(* CoDeSys 2.3 project: CX_KNX_TEST.pro *)
(* Title: BC and KL6301 *)
(* Version: 1.00 *)
(* Author: RV *)
(* Description: Demoproject for receive EIB Data
BC9000
KL6301
KL9010 *)
(* Libraries: TcpIp.lib 13.10.11 10:31:34, TcUtilities.lib 8.2.10 17:42:18, TcSocketHelper.lib 20.8.09 10:46:08, TcBase.lib 14.5.09 12:14:08, standard.lib 5.6.98 12:03:02, ClientStrSock.lib 19.10.12 18:01:27, TcSystem.lib 9.3.10 11:21:30, TcModbusSrv.lib 26.1.12 11:11:48, TcKL6301.lib 4.11.10 11:26:24 *)

(* Task configuration *)
TASK NeueTask (PRIORITY := 0, INTERVAL := T#10ms);
	MAIN();
END_TASK
TASK PowerCalc (PRIORITY := 2, INTERVAL := T#100ms);
	CalcPower();
END_TASK
TASK AdsSend (PRIORITY := 3, INTERVAL := T#1000ms);
	CheckLight();
END_TASK
TASK NewTask (PRIORITY := 1, INTERVAL := T#250ms);
	POWER_OFF_TEST();
	ReadADS();
END_TASK

(* Global variable list: Global_Variables_Power *)
VAR_GLOBAL

	KL3403_ctrl_1 AT%Q* : BYTE;

	KL3403_1_P1 AT%I* : INT;
	KL3403_1_P2 AT%I* : INT;
	KL3403_1_P3 AT%I* : INT;

	KL3403_1_P: REAL;
	KL3403_1_V: REAL;
	KL3403_1_I: REAL;

	KL3403_2_P1 AT%I* : INT;
	KL3403_2_P2 AT%I* : INT;
	KL3403_2_P3 AT%I* : INT;

	KL3403_2_P: REAL;
	KL3403_2_V: REAL;
	KL3403_2_I: REAL;

	KL3403_3_P1 AT%I* : INT;
	KL3403_3_P2 AT%I* : INT;
	KL3403_3_P3 AT%I* : INT;

	KL3403_3_P: REAL;
	KL3403_3_V: REAL;
	KL3403_3_I: REAL;

	KL3403_4_P1 AT%I* : INT;
	KL3403_4_P2 AT%I* : INT;
	KL3403_4_P3 AT%I* : INT;

	KL3403_4_P: REAL;
	KL3403_4_V: REAL;
	KL3403_4_I: REAL;

	KL3403_5_P1 AT%I* : INT;
	KL3403_5_P2 AT%I* : INT;
	KL3403_5_P3 AT%I* : INT;

	KL3403_5_P: REAL;
	KL3403_5_V: REAL;
	KL3403_5_I: REAL;

(*array of powers in VRU*)

(*
1 - schavp1		3
2 - schrd			11
3 - parouvl		2
4 - schnvd		5
5 - schrb			6
6 - schl			9
7 - schrov		1
8 - schss			10
9 - schuf			4
10 - schno		7
11 - hammam		8

7 - schrov		1
3 - parouvl		2
1 - schavp1		3
9 - schuf			4
4 - schnvd		5
5 - schrb			6
10 - schno		7
11 - hammam		8
6 - schl			9
8 - schss			10
2 - schrd			11

*)

	POWER_LIMIT: REAL;
	Current_switch_pos: INT;

	power_VRU_switch:  ARRAY[1..11] OF BOOL;
	(* priority*)
	power_VRU_address:  ARRAY[1..11] OF EIB_GROUP_ADDR;
	power_VRU_value: ARRAY[1..11] OF REAL;


	PowerSystemSwitcher: BOOL := TRUE;

END_VAR

(* Global variable list: Globale_Variablen *)
VAR_GLOBAL
    	bCloseAll 					: BOOL := TRUE;
   	bCreateSock					: BOOL := TRUE;

	ModByte			: BYTE;
	ModbusVentili	: BYTE;

	OutLightBytes		: BYTE;
	ControlLights		: BYTE;

	SCHAV			: ARRAY [1..4] OF INT;
	SCHNOG		: ARRAY [1..9] OF BOOL;

	schav_receive_stack AT %MB500 : ARRAY[1..7] OF INT;
	schav_force_stack AT %MB250 : ARRAY[1..7] OF INT;
	schnog_receive_stack AT %MB65 : ARRAY[1..19] OF BOOL;
	schnog_force_stack AT %MB265 : ARRAY[1..19] OF BOOL;
	schszp_receive_stack AT %MB100 : ARRAY[1..116] OF BOOL;
	schszp_force_stack AT %MB4500 : ARRAY[1..116] OF BOOL;
	(*tempMain_udp_packet AT %MB6000 : Udp_Packet;*)
	Main_udp_packet AT %MB2000 : Udp_Packet;
	Force_udp_packet AT %MB3000 : Udp_Packet;
	Temp_of_int AT %MB3006 : ARRAY[1..213] OF INT; (*область памяти совпадает с Force_udp_packet*)
	Confirmation_packet : Udp_Confirm;
	Received_packet AT %MB750 : Udp_Confirm;

	RESET_Edge : BOOL:=FALSE;
	TestWord : WORD;

	rByte : DINT;
	bSendConf : BOOL := FALSE;
	PacketSize: INT;
	Checksum_send : WORD;
	Checksum_incom : WORD;

	value3: INT;
	value2: INT;

	(*Считываем занчения вентиляторов*)
	CoolerByte		: BYTE;

	(* EIB terminal KL6301 process data 24 Byte input and 24 Byte output data K-Bus*)
	ShNOG_Garage_OG_22 AT %MB4 : BOOL:=FALSE;  (*Передаваемый параметр на другой контроллер. Свет в гараже - фуекция неисправного выхода модуля ABB KNX*)
	ShAV_Vent_V3 AT %MB5 : BOOL:=FALSE;  (*Передаваемый параметр на другой контроллер. Свет в туалете*)
	LightLandscape	: BOOL:=FALSE;  (*Передаваемый параметр на другой контроллер. Свет ландшафта*)
	LightNight AT %MB6 : BOOL := FALSE;  (*Передаваемый параметр на другой контроллер. "Ночь"*)
	KNXISDAY : BOOL := FALSE;
	KNXISTWILIGHT : BOOL := FALSE;
	LightNight_Clock AT %MB8 : BOOL := FALSE;

	SystemTime AT %MB4000 : TIMESTRUCT;
(*
	SS_H_AUT : WORD := 17; (*17*)
	SR_H_AUT : WORD := 6;
	SS_M_AUT : WORD := 19; (*19*)
	SR_M_AUT : WORD := 59;
	SS_H_WIN : WORD := 17; (*16*)
	SR_H_WIN : WORD := 8;
	SS_M_WIN : WORD := 19;
	SR_M_WIN : WORD := 29;
	SS_H_SPR : WORD := 19;
	SR_H_SPR : WORD := 5;
	SS_M_SPR : WORD := 19;
	SR_M_SPR : WORD := 29;
	SS_H_SUM : WORD := 21;
	SR_H_SUM : WORD := 4;
	SS_M_SUM : WORD := 01;
	SR_M_SUM : WORD := 01;
*)

	SS_H_JAN : WORD := 16;
	SR_H_JAN : WORD := 9;
	SS_M_JAN : WORD := 8;
	SR_M_JAN : WORD := 0;
	SS_H_FEB : WORD := 17;
	SR_H_FEB : WORD := 8;
	SS_M_FEB : WORD := 3;
	SR_M_FEB : WORD := 25;
	SS_H_MAR : WORD := 18;
	SR_H_MAR : WORD := 7;
	SS_M_MAR : WORD := 4;
	SR_M_MAR : WORD := 23;
	SS_H_APR : WORD := 19;
SR_H_APR : WORD := 6;
	SS_M_APR : WORD := 7;
SR_M_APR : WORD := 2;
	SS_H_MAY : WORD := 20;
SR_H_MAY : WORD := 4;
SS_M_MAY : WORD := 7;
SR_M_MAY : WORD := 48;
SS_H_JUN : WORD := 21;
SR_H_JUN : WORD := 3;
SS_M_JUN : WORD := 3;
SR_M_JUN : WORD := 55;
SS_H_JUL : WORD := 21;
SR_H_JUL : WORD := 3;
SS_M_JUL : WORD := 18;
SR_M_JUL : WORD := 51;
SS_H_AUG : WORD := 20;
SR_H_AUG : WORD := 4;
SS_M_AUG : WORD := 39;
SR_M_AUG : WORD := 35;
SS_H_SEP : WORD := 19;
SR_H_SEP : WORD := 5;
SS_M_SEP : WORD := 27;
SR_M_SEP : WORD := 35;
SS_H_OCT : WORD := 18;
SR_H_OCT : WORD := 6;
SS_M_OCT : WORD := 8;
SR_M_OCT : WORD := 33;
SS_H_NOV : WORD := 16;
SR_H_NOV : WORD := 7;
SS_M_NOV : WORD := 52;
SR_M_NOV : WORD := 36;
SS_H_DEC : WORD := 16;
SR_H_DEC : WORD := 8;
SS_M_DEC : WORD := 4;
SR_M_DEC : WORD := 36;

	JAN : WORD := 1;
	FEB : WORD := 2;
	MAR : WORD := 3;
	APR : WORD := 4;
	MAY : WORD := 5;
	JUN : WORD := 6;
	JUL : WORD := 7;
	AUG : WORD := 8;
	SEP : WORD := 9;
	OCT : WORD := 10;
	NOV : WORD := 11;
	DEC : WORD := 12;

	KNX_BRIGHTNESS_L : DINT;
	KNX_BRIGHTNESS_C : DINT;
	KNX_BRIGHTNESS_R : DINT;

	LightGarageSecurity : BOOL := FALSE;
	LightGatesLight AT %MB7 : BOOL:=FALSE;  (*Передаваемый параметр на другой контроллер. Выключатель света ворот в комнате охраны*)


	ADSSend: BOOL:=FALSE;

	KL6301_IN_0 AT %IB0: ARRAY[1..24] OF BYTE;
	KL6301_OUT_0 AT %QB0: ARRAY[1..24] OF BYTE;
	Taster0_LUX: BOOL;
	Taster1_LUX: BOOL;
	Taster2_LUX: BOOL;
	Taster3_LUX: BOOL;

	AllOff: BOOL;

	KoefV: BOOL:=FALSE;
	KoefI: BOOL:=FALSE;
	KoefP: BOOL:=TRUE;

	garage_OG_1: BOOL;
	garage_OG_2: BOOL;
	garage_OG_3: BOOL;
	garage_OG_4: BOOL;
	garage_OG_5: BOOL;
	garage_OG_6: BOOL;
	garage_OG_7: BOOL;
	garage_OG_8: BOOL;
	garage_OG_9: BOOL;
	garage_OG_10: BOOL;
	garage_OG_11: BOOL;
	garage_OG_12: BOOL;
	garage_OG_13: BOOL;
	garage_OG_14: BOOL;
	garage_OG_15: BOOL;
	garage_OG_16: BOOL;
	garage_OG_17: BOOL;
	garage_OG_18: BOOL;
	garage_OG_19: BOOL;
	garage_OG_20: BOOL;
	garage_OG_21: BOOL;
	garage_OG_22: BOOL;
	garage_OG_23: BOOL;
	garage_OG_24: BOOL;
	garage_OG_25: BOOL;
	garage_OG_26: BOOL;
	garage_OG_27: BOOL;
	garage_OG_28: BOOL;
	garage_OG_29: BOOL;

	SHUF_PRESSED: BOOL:= FALSE;

	DATA_SCALE_H									:INT :=255;
	DATA_SCALE_L									:INT :=0;
	DATA_SCALE_H_FAN								:INT :=32000;
	DATA_SCALE_L_FAN								:INT :=0;


END_VAR

VAR_GLOBAL CONSTANT
        TCPADS_MAXUDP_BUFFSIZE : UDINT :=32000;
END_VAR

(* Global variable list: Globale_Variablen_EIB *)
VAR_GLOBAL
	EIB_DATA_READ:  ARRAY[1..14] OF BYTE;
	Lux_REAL: REAL;	(* LUX *)
	Switch_0: BOOL;	(* Switch 1/2/1*)
	Switch_1: BOOL;	(* Switch 1/2/2*)
	Taster_0 AT %QX32.0: BOOL;
	Taster_1 AT %QX32.1: BOOL;
	Temp_0_KL3312 AT %IB26:INT;
	Temp_1_KL3312 AT %IB30:INT;
	IN_0_KL1012 AT %IX32.0:BOOL;
	IN_1_KL1012 AT %IX32.1:BOOL;
	str_Send: EIB_SEND;
	EIB_4FachT: BOOL;
	ToggleBit: BOOL;
	Soll_Lamp_Dimmer: INT;

	TurnAllTheLight: BOOL := FALSE;
END_VAR

(* Global variable list: TwinCAT_Configuration *)
(* Generated automatically by TwinCAT - (read only) *)
VAR_CONFIG
	.KL3403_ctrl_1 AT %QB36 : BYTE;	(*  ~ {LinkedWith:TIID^Device 3 (CX1100)^CX1100-KB^Term 2 (KL3403)^Channel 2^Ctrl;TIID^Device 3 (CX1100)^CX1100-KB^Term 2 (KL3403)^Channel 3^Ctrl;TIID^Device 3 (CX1100)^CX1100-KB^Term 3 (KL3403)^Channel 1^Ctrl;TIID^Device 3 (CX1100)^CX1100-KB^Term 3 (KL3403)^Channel 2^Ctrl;TIID^Device 3 (CX1100)^CX1100-KB^Term 3 (KL3403)^Channel 3^Ctrl;TIID^Device 3 (CX1100)^CX1100-KB^Term 4 (KL3403)^Channel 1^Ctrl;TIID^Device 3 (CX1100)^CX1100-KB^Term 4 (KL3403)^Channel 2^Ctrl;TIID^Device 3 (CX1100)^CX1100-KB^Term 4 (KL3403)^Channel 3^Ctrl;TIID^Device 3 (CX1100)^CX1100-KB^Term 5 (KL3403)^Channel 1^Ctrl;TIID^Device 3 (CX1100)^CX1100-KB^Term 5 (KL3403)^Channel 2^Ctrl;TIID^Device 3 (CX1100)^CX1100-KB^Term 5 (KL3403)^Channel 3^Ctrl;TIID^Device 3 (CX1100)^CX1100-KB^Term 6 (KL3403)^Channel 1^Ctrl;TIID^Device 3 (CX1100)^CX1100-KB^Term 6 (KL3403)^Channel 2^Ctrl;TIID^Device 3 (CX1100)^CX1100-KB^Term 6 (KL3403)^Channel 3^Ctrl;TIID^Device 3 (CX1100)^CX1100-KB^Term 2 (KL3403)^Channel 1^Ctrl} *)
	.KL3403_1_P1 AT %IB36 : INT;	(*  ~ {LinkedWith:TIID^Device 3 (CX1100)^CX1100-KB^Term 2 (KL3403)^Channel 1^Data In} *)
	.KL3403_1_P2 AT %IB38 : INT;	(*  ~ {LinkedWith:TIID^Device 3 (CX1100)^CX1100-KB^Term 2 (KL3403)^Channel 2^Data In} *)
	.KL3403_1_P3 AT %IB40 : INT;	(*  ~ {LinkedWith:TIID^Device 3 (CX1100)^CX1100-KB^Term 2 (KL3403)^Channel 3^Data In} *)
	.KL3403_2_P1 AT %IB42 : INT;	(*  ~ {LinkedWith:TIID^Device 3 (CX1100)^CX1100-KB^Term 3 (KL3403)^Channel 1^Data In} *)
	.KL3403_2_P2 AT %IB44 : INT;	(*  ~ {LinkedWith:TIID^Device 3 (CX1100)^CX1100-KB^Term 3 (KL3403)^Channel 2^Data In} *)
	.KL3403_2_P3 AT %IB46 : INT;	(*  ~ {LinkedWith:TIID^Device 3 (CX1100)^CX1100-KB^Term 3 (KL3403)^Channel 3^Data In} *)
	.KL3403_3_P1 AT %IB48 : INT;	(*  ~ {LinkedWith:TIID^Device 3 (CX1100)^CX1100-KB^Term 4 (KL3403)^Channel 1^Data In} *)
	.KL3403_3_P2 AT %IB50 : INT;	(*  ~ {LinkedWith:TIID^Device 3 (CX1100)^CX1100-KB^Term 4 (KL3403)^Channel 2^Data In} *)
	.KL3403_3_P3 AT %IB52 : INT;	(*  ~ {LinkedWith:TIID^Device 3 (CX1100)^CX1100-KB^Term 4 (KL3403)^Channel 3^Data In} *)
	.KL3403_4_P1 AT %IB54 : INT;	(*  ~ {LinkedWith:TIID^Device 3 (CX1100)^CX1100-KB^Term 5 (KL3403)^Channel 1^Data In} *)
	.KL3403_4_P2 AT %IB56 : INT;	(*  ~ {LinkedWith:TIID^Device 3 (CX1100)^CX1100-KB^Term 5 (KL3403)^Channel 2^Data In} *)
	.KL3403_4_P3 AT %IB58 : INT;	(*  ~ {LinkedWith:TIID^Device 3 (CX1100)^CX1100-KB^Term 5 (KL3403)^Channel 3^Data In} *)
	.KL3403_5_P1 AT %IB60 : INT;	(*  ~ {LinkedWith:TIID^Device 3 (CX1100)^CX1100-KB^Term 6 (KL3403)^Channel 1^Data In} *)
	.KL3403_5_P2 AT %IB62 : INT;	(*  ~ {LinkedWith:TIID^Device 3 (CX1100)^CX1100-KB^Term 6 (KL3403)^Channel 2^Data In} *)
	.KL3403_5_P3 AT %IB64 : INT;	(*  ~ {LinkedWith:TIID^Device 3 (CX1100)^CX1100-KB^Term 6 (KL3403)^Channel 3^Data In} *)
END_VAR

(* Data type *)
TYPE ST_FifoEntry :
STRUCT
	sRemoteHost		: STRING(15);		(* Remote address. String containing an (Ipv4) Internet Protocol dotted address. *)
	nRemotePort		: UDINT;			(* Remote Internet Protocol (IP) port. *)
	msg				: STRING;			(* Udp packet data *)
END_STRUCT
END_TYPE

(* Data type *)
TYPE Udp_Confirm :
STRUCT
	title_packet_num : INT;
	title_packet_code : INT;
	title_packet_crc : INT;
	data_pointer : INT;
	data_new_value : INT;
END_STRUCT
END_TYPE

(* Data type *)
TYPE Udp_Packet :
STRUCT
	title_packet_num : INT;
	title_packet_code : INT;
	title_packet_crc : INT;
	grsch_P : ARRAY[1..5] OF INT;
	grsch_V : ARRAY[1..5] OF INT;
	grsch_I : ARRAY[1..5] OF INT;
	grsch_garage_og : ARRAY[1..29] OF INT;
	grsch_power_VRU_value : ARRAY[1..11] OF INT;
	grsch_power_limit : INT;
	grsch_current_switch_pos : INT;
	grsch_power_VRU_switch : ARRAY[1..11] OF INT;
	grsch_SHUF_PRESSED : INT;
	grsch_power_system_switcher : INT;
	schav_stack : ARRAY[1..7] OF INT;
	schnog_stack : ARRAY[1..19] OF INT;
	schszp_stack  : ARRAY[1..116] OF INT;
END_STRUCT
END_TYPE

(* POU MAIN, ST *)
PROGRAM MAIN
VAR

	fbReadCoils : FB_MBReadCoils;
	bReadCoils : BOOL;
	nValue : BYTE;


	(* CX Controller *)
	(* KL6301 *)
	(* KL2xx2 *)
	(* KL9010 *)
	(* 1. EIB Device 2 Channel Switch Group Address 1/2/1 and 1 /2/2 *)
	(* 2. EIB Device Lux meter Group Address 1/1/5 *)
	fb_KL6301_0 : KL6301;	(* EIB functonblock *)
	i: INT := 0;				(* CASE *)
	EIB_DATA_SEND_0: EIB_SEND_DATA;
	fbTimer_0: TON;
	TimerOn: BOOL := FALSE;
	FLAG_01: BOOL := TRUE;
END_VAR
CASE i OF
0: 	fb_KL6301_0.bActivate :=FALSE; (*Start EIB Functionblock*)
	i := 1;

1:	fb_KL6301_0.EIB_PHYS_ADDR.Area:=2;		(* EIB Address 2.3.4 *)
	fb_KL6301_0.EIB_PHYS_ADDR.Line:=3;
	fb_KL6301_0.EIB_PHYS_ADDR.Device:=4;
	(* Filter 1 1/1/0 LEN 63*)
	fb_KL6301_0.EIB_GROUP_FILTER[1].GROUP_ADDR.MAIN:=1;
	fb_KL6301_0.EIB_GROUP_FILTER[1].GROUP_ADDR.SUB_MAIN:=1;
	fb_KL6301_0.EIB_GROUP_FILTER[1].GROUP_ADDR.NUMBER:=0;
	fb_KL6301_0.EIB_GROUP_FILTER[1].GROUP_LEN:=63;

	fb_KL6301_0.EIB_GROUP_FILTER[2].GROUP_ADDR.MAIN:=3;
	fb_KL6301_0.EIB_GROUP_FILTER[2].GROUP_ADDR.SUB_MAIN:=1;
	fb_KL6301_0.EIB_GROUP_FILTER[2].GROUP_ADDR.NUMBER:=0;
	fb_KL6301_0.EIB_GROUP_FILTER[2].GROUP_LEN:=63;

	fb_KL6301_0.EIB_GROUP_FILTER[3].GROUP_ADDR.MAIN:=5;
	fb_KL6301_0.EIB_GROUP_FILTER[3].GROUP_ADDR.SUB_MAIN:=1;
	fb_KL6301_0.EIB_GROUP_FILTER[3].GROUP_ADDR.NUMBER:=0;
	fb_KL6301_0.EIB_GROUP_FILTER[3].GROUP_LEN:=63;

	fb_KL6301_0.bActivate :=TRUE; (*Start EIB Functionblock*)

	IF fb_KL6301_0.bReady THEN
		IF NOT fb_KL6301_0.bError THEN
			i:=2;  (* EIB functionblock is now ready to send and receive *)
		ELSE
			i:=100; (* EIB ERROR*)
		END_IF
	END_IF
2:
(*Соберем всю инфу. По крайней мере, попробуем *)
KNX_Init;
(*POWER_OFF_TEST;*)

100:	;(*ERROR EIB*)
END_CASE

fb_KL6301_0(
	idx:=20,
	KL6301_IN:=KL6301_IN_0,				(* Terminal variable - address IN *)
	KL6301_OUT:=KL6301_OUT_0 );			(* Terminal variable - address OUT *)

Main_EIB_REC;

IF KoefV=TRUE THEN
	KL3403_ctrl_1:=1;
	KoefI:=FALSE;
	KoefV:=FALSE;
	KoefP:=FALSE;

END_IF

IF KoefI=TRUE THEN
	KL3403_ctrl_1:=0;
	KoefI:=FALSE;
	KoefV:=FALSE;
	KoefP:=FALSE;
END_IF

IF KoefP=TRUE THEN
	KL3403_ctrl_1:=2;
	KoefI:=FALSE;
	KoefV:=FALSE;
	KoefP:=FALSE;
END_IF

IF SHUF_PRESSED = TRUE THEN
	POWER_OFF_TEST;
	SHUF_PRESSED:= FALSE;
END_IF;

(* ZAPLATKA ZIMA VESNA LETO OSEN *)

IF (SystemTime.wMonth = JAN) AND SystemTime.wHour = SS_H_JAN AND SystemTime.wMinute = SS_M_JAN THEN
	LightNight_Clock := TRUE;						
END_IF;							
IF (SystemTime.wMonth = JAN) AND SystemTime.wHour = SR_H_JAN AND SystemTime.wMinute = SR_M_JAN THEN							
	LightNight_Clock := FALSE;						
END_IF;							
IF (SystemTime.wMonth = FEB) AND SystemTime.wHour = SS_H_FEB AND SystemTime.wMinute = SS_M_FEB THEN							
	LightNight_Clock := TRUE;						
END_IF;							
IF (SystemTime.wMonth = FEB) AND SystemTime.wHour = SR_H_FEB AND SystemTime.wMinute = SR_M_FEB THEN							
	LightNight_Clock := FALSE;						
END_IF;							
IF (SystemTime.wMonth = MAR) AND SystemTime.wHour = SS_H_MAR AND SystemTime.wMinute = SS_M_MAR THEN							
	LightNight_Clock := TRUE;						
END_IF;							
IF (SystemTime.wMonth = MAR) AND SystemTime.wHour = SR_H_MAR AND SystemTime.wMinute = SR_M_MAR THEN							
	LightNight_Clock := FALSE;						
END_IF;							
IF (SystemTime.wMonth = APR) AND SystemTime.wHour = SS_H_APR AND SystemTime.wMinute = SS_M_APR THEN							
	LightNight_Clock := TRUE;						
END_IF;							
IF (SystemTime.wMonth = APR) AND SystemTime.wHour = SR_H_APR AND SystemTime.wMinute = SR_M_APR THEN							
	LightNight_Clock := FALSE;						
END_IF;							
IF (SystemTime.wMonth = MAY) AND SystemTime.wHour = SS_H_MAY AND SystemTime.wMinute = SS_M_MAY THEN							
	LightNight_Clock := TRUE;						
END_IF;							
IF (SystemTime.wMonth = MAY) AND SystemTime.wHour = SR_H_MAY AND SystemTime.wMinute = SR_M_MAY THEN							
	LightNight_Clock := FALSE;						
END_IF;							
IF (SystemTime.wMonth = JUN) AND SystemTime.wHour = SS_H_JUN AND SystemTime.wMinute = SS_M_JUN THEN							
	LightNight_Clock := TRUE;						
END_IF;							
IF (SystemTime.wMonth = JUN) AND SystemTime.wHour = SR_H_JUN AND SystemTime.wMinute = SR_M_JUN THEN							
	LightNight_Clock := FALSE;						
END_IF;							
IF (SystemTime.wMonth = JUL) AND SystemTime.wHour = SS_H_JUL AND SystemTime.wMinute = SS_M_JUL THEN							
	LightNight_Clock := TRUE;						
END_IF;							
IF (SystemTime.wMonth = JUL) AND SystemTime.wHour = SR_H_JUL AND SystemTime.wMinute = SR_M_JUL THEN							
	LightNight_Clock := FALSE;						
END_IF;							
IF (SystemTime.wMonth = AUG) AND SystemTime.wHour = SS_H_AUG AND SystemTime.wMinute = SS_M_AUG THEN							
	LightNight_Clock := TRUE;						
END_IF;							
IF (SystemTime.wMonth = AUG) AND SystemTime.wHour = SR_H_AUG AND SystemTime.wMinute = SR_M_AUG THEN							
	LightNight_Clock := FALSE;						
END_IF;							
IF (SystemTime.wMonth = SEP) AND SystemTime.wHour = SS_H_SEP AND SystemTime.wMinute = SS_M_SEP THEN							
	LightNight_Clock := TRUE;						
END_IF;							
IF (SystemTime.wMonth = SEP) AND SystemTime.wHour = SR_H_SEP AND SystemTime.wMinute = SR_M_SEP THEN							
	LightNight_Clock := FALSE;						
END_IF;							
IF (SystemTime.wMonth = OCT) AND SystemTime.wHour = SS_H_OCT AND SystemTime.wMinute = SS_M_OCT THEN							
	LightNight_Clock := TRUE;						
END_IF;							
IF (SystemTime.wMonth = OCT) AND SystemTime.wHour = SR_H_OCT AND SystemTime.wMinute = SR_M_OCT THEN							
	LightNight_Clock := FALSE;						
END_IF;							
IF (SystemTime.wMonth = NOV) AND SystemTime.wHour = SS_H_NOV AND SystemTime.wMinute = SS_M_NOV THEN							
	LightNight_Clock := TRUE;						
END_IF;							
IF (SystemTime.wMonth = NOV) AND SystemTime.wHour = SR_H_NOV AND SystemTime.wMinute = SR_M_NOV THEN							
	LightNight_Clock := FALSE;						
END_IF;							
IF (SystemTime.wMonth = DEC) AND SystemTime.wHour = SS_H_DEC AND SystemTime.wMinute = SS_M_DEC THEN							
	LightNight_Clock := TRUE;						
END_IF;							
IF (SystemTime.wMonth = DEC) AND SystemTime.wHour = SR_H_DEC AND SystemTime.wMinute = SR_M_DEC THEN
	LightNight_Clock := FALSE;
END_IF;

(*
IF (SystemTime.wMonth = DEC OR SystemTime.wMonth = JAN OR SystemTime.wMonth = FEB) AND SystemTime.wHour = SS_H_WIN AND SystemTime.wMinute = SS_M_WIN THEN
	LightNight_Clock := TRUE;
END_IF;
IF (SystemTime.wMonth = DEC OR SystemTime.wMonth = JAN OR SystemTime.wMonth = FEB) AND SystemTime.wHour = SR_H_WIN AND SystemTime.wMinute = SR_M_WIN THEN
	LightNight_Clock := FALSE;
END_IF;

IF (SystemTime.wMonth = MAR OR SystemTime.wMonth = APR OR SystemTime.wMonth = MAY) AND SystemTime.wHour = SS_H_SPR AND SystemTime.wMinute = SS_M_SPR THEN
	LightNight_Clock := TRUE;
END_IF;
IF (SystemTime.wMonth = MAR OR SystemTime.wMonth = APR OR SystemTime.wMonth = MAY) AND SystemTime.wHour = SR_H_SPR AND SystemTime.wMinute = SR_M_SPR THEN
	LightNight_Clock := FALSE;
END_IF;

IF (SystemTime.wMonth = JUN OR SystemTime.wMonth = JUL OR SystemTime.wMonth = AUG) AND SystemTime.wHour = SS_H_SUM AND SystemTime.wMinute = SS_M_SUM THEN
	LightNight_Clock := TRUE;
END_IF;
IF (SystemTime.wMonth = JUN OR SystemTime.wMonth = JUL OR SystemTime.wMonth = AUG) AND SystemTime.wHour = SR_H_SUM AND SystemTime.wMinute = SR_M_SUM THEN
	LightNight_Clock := FALSE;
END_IF;

IF (SystemTime.wMonth = SEP OR SystemTime.wMonth = OCT OR SystemTime.wMonth = NOV) AND SystemTime.wHour = SS_H_AUT AND SystemTime.wMinute = SS_M_AUT THEN
	LightNight_Clock := TRUE;
END_IF;
IF (SystemTime.wMonth = SEP OR SystemTime.wMonth = OCT OR SystemTime.wMonth = NOV) AND SystemTime.wHour = SR_H_AUT AND SystemTime.wMinute = SR_M_AUT THEN
	LightNight_Clock := FALSE;
END_IF;

ZAPLATKA *)

IF KL6301_IN_0[10] = 16#0081 THEN
	LightGatesLight := TRUE;
ELSE
	LightGatesLight := FALSE;
END_IF;

Udp_send_packet_init;
PeerToPeer;
Udp_receive_packet_init;

IF (SystemTime.wDay = 15) AND SystemTime.wHour = 4 AND SystemTime.wMinute = 00 THEN
RESET_Edge:= TRUE;
AutoReset;
END_IF;
END_PROGRAM

(* POU KNX_Init, CFC *)
PROGRAM KNX_Init
VAR

(*свет*)
	Group_1_1_1: EIB_GROUP_ADDR := (MAIN:=1,SUB_MAIN:=1,NUMBER:=1);
	Group_1_1_2: EIB_GROUP_ADDR := (MAIN:=1,SUB_MAIN:=1,NUMBER:=2);
	Group_1_1_3: EIB_GROUP_ADDR := (MAIN:=1,SUB_MAIN:=1,NUMBER:=3);
	Group_1_1_4: EIB_GROUP_ADDR := (MAIN:=1,SUB_MAIN:=1,NUMBER:=4);
	Group_1_1_5: EIB_GROUP_ADDR := (MAIN:=1,SUB_MAIN:=1,NUMBER:=5);
	Group_1_1_6: EIB_GROUP_ADDR := (MAIN:=1,SUB_MAIN:=1,NUMBER:=6);
	Group_1_1_7: EIB_GROUP_ADDR := (MAIN:=1,SUB_MAIN:=1,NUMBER:=7);
	Group_1_1_8: EIB_GROUP_ADDR := (MAIN:=1,SUB_MAIN:=1,NUMBER:=8);
	Group_1_1_9: EIB_GROUP_ADDR := (MAIN:=1,SUB_MAIN:=1,NUMBER:=9);
	Group_1_1_10: EIB_GROUP_ADDR := (MAIN:=1,SUB_MAIN:=1,NUMBER:=10);
	Group_1_1_11: EIB_GROUP_ADDR := (MAIN:=1,SUB_MAIN:=1,NUMBER:=11);
	Group_1_1_12: EIB_GROUP_ADDR := (MAIN:=1,SUB_MAIN:=1,NUMBER:=12);
	Group_1_1_13: EIB_GROUP_ADDR := (MAIN:=1,SUB_MAIN:=1,NUMBER:=13);
	Group_1_1_14: EIB_GROUP_ADDR := (MAIN:=1,SUB_MAIN:=1,NUMBER:=14);
	Group_1_1_15: EIB_GROUP_ADDR := (MAIN:=1,SUB_MAIN:=1,NUMBER:=15);
	Group_1_1_16: EIB_GROUP_ADDR := (MAIN:=1,SUB_MAIN:=1,NUMBER:=16);
	Group_1_1_17: EIB_GROUP_ADDR := (MAIN:=1,SUB_MAIN:=1,NUMBER:=17);
	Group_1_1_18: EIB_GROUP_ADDR := (MAIN:=1,SUB_MAIN:=1,NUMBER:=18);
	Group_1_1_19: EIB_GROUP_ADDR := (MAIN:=1,SUB_MAIN:=1,NUMBER:=19);
	Group_1_1_20: EIB_GROUP_ADDR := (MAIN:=1,SUB_MAIN:=1,NUMBER:=20);
	Group_1_1_21: EIB_GROUP_ADDR := (MAIN:=1,SUB_MAIN:=1,NUMBER:=21);
	Group_1_1_22: EIB_GROUP_ADDR := (MAIN:=1,SUB_MAIN:=1,NUMBER:=22);
	Group_1_1_23: EIB_GROUP_ADDR := (MAIN:=1,SUB_MAIN:=1,NUMBER:=23);
	Group_1_1_24: EIB_GROUP_ADDR := (MAIN:=1,SUB_MAIN:=1,NUMBER:=24);
	Group_1_1_25: EIB_GROUP_ADDR := (MAIN:=1,SUB_MAIN:=1,NUMBER:=25);
	Group_1_1_26: EIB_GROUP_ADDR := (MAIN:=1,SUB_MAIN:=1,NUMBER:=26);
	Group_1_1_27: EIB_GROUP_ADDR := (MAIN:=1,SUB_MAIN:=1,NUMBER:=27);
	Group_1_1_28: EIB_GROUP_ADDR := (MAIN:=1,SUB_MAIN:=1,NUMBER:=28);
	Group_1_1_29: EIB_GROUP_ADDR := (MAIN:=1,SUB_MAIN:=1,NUMBER:=29);
	Group_1_1_30: EIB_GROUP_ADDR := (MAIN:=1,SUB_MAIN:=1,NUMBER:=30);
	Group_1_1_31: EIB_GROUP_ADDR := (MAIN:=1,SUB_MAIN:=1,NUMBER:=31);
	Group_1_1_32: EIB_GROUP_ADDR := (MAIN:=1,SUB_MAIN:=1,NUMBER:=32);
	Group_1_1_33: EIB_GROUP_ADDR := (MAIN:=1,SUB_MAIN:=1,NUMBER:=33);
	Group_1_1_34: EIB_GROUP_ADDR := (MAIN:=1,SUB_MAIN:=1,NUMBER:=34);
	Group_1_1_35: EIB_GROUP_ADDR := (MAIN:=1,SUB_MAIN:=1,NUMBER:=35);
	Group_1_1_36: EIB_GROUP_ADDR := (MAIN:=1,SUB_MAIN:=1,NUMBER:=36);
	Group_1_1_37: EIB_GROUP_ADDR := (MAIN:=1,SUB_MAIN:=1,NUMBER:=37);
	Group_1_1_38: EIB_GROUP_ADDR := (MAIN:=1,SUB_MAIN:=1,NUMBER:=38);
	KNXSYSTEM_WEATHERST_BRIGHTNES_L: EIB_GROUP_ADDR := (MAIN:=5,SUB_MAIN:=1,NUMBER:=2);
	KNXSYSTEM_WEATHERST_BRIGHTNES_C: EIB_GROUP_ADDR := (MAIN:=5,SUB_MAIN:=1,NUMBER:=3);
	KNXSYSTEM_WEATHERST_BRIGHTNES_R: EIB_GROUP_ADDR := (MAIN:=5,SUB_MAIN:=1,NUMBER:=4);
	KNXSYSTEM_WEATHERST_ISDAY: EIB_GROUP_ADDR := (MAIN:=5,SUB_MAIN:=1,NUMBER:=6);
	KNXSYSTEM_WEATHERST_ISTWILIGHT: EIB_GROUP_ADDR := (MAIN:=5,SUB_MAIN:=1,NUMBER:=40);

	init1: EIB_READ_SEND;
	init2: EIB_READ_SEND;
	init4: EIB_READ_SEND;
	init3: EIB_READ_SEND;
	init5: EIB_READ_SEND;
	init6: EIB_READ_SEND;
	init7: EIB_READ_SEND;
	init8: EIB_READ_SEND;
	init9: EIB_READ_SEND;
	init10: EIB_READ_SEND;
	init11: EIB_READ_SEND;
	init12: EIB_READ_SEND;
	init24: EIB_READ_SEND;
	init23: EIB_READ_SEND;
	init22: EIB_READ_SEND;
	init21: EIB_READ_SEND;
	init20: EIB_READ_SEND;
	init19: EIB_READ_SEND;
	init13: EIB_READ_SEND;
	init14: EIB_READ_SEND;
	init15: EIB_READ_SEND;
	init16: EIB_READ_SEND;
	init17: EIB_READ_SEND;
	init18: EIB_READ_SEND;
	init25: EIB_READ_SEND;
	init26: EIB_READ_SEND;
	init27: EIB_READ_SEND;
	init28: EIB_READ_SEND;
	init29: EIB_READ_SEND;
	init30: EIB_READ_SEND;
	init31: EIB_READ_SEND;
	init32: EIB_READ_SEND;
	init33: EIB_READ_SEND;
	init34: EIB_READ_SEND;
	init35: EIB_READ_SEND;
	init36: EIB_READ_SEND;
	init37: EIB_READ_SEND;
	init38: EIB_READ_SEND;
	init39: EIB_READ_SEND;
	init40: EIB_READ_SEND;
	init41: EIB_READ_SEND;
	init42: EIB_READ_SEND;
	init43: EIB_READ_SEND;
END_VAR
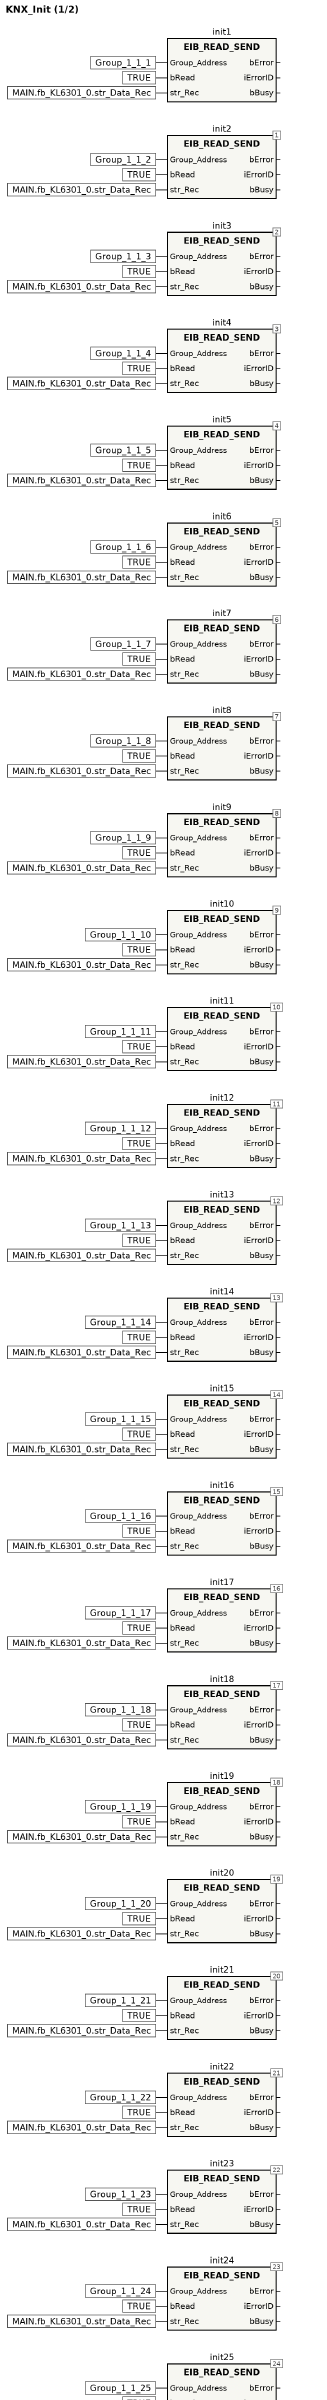
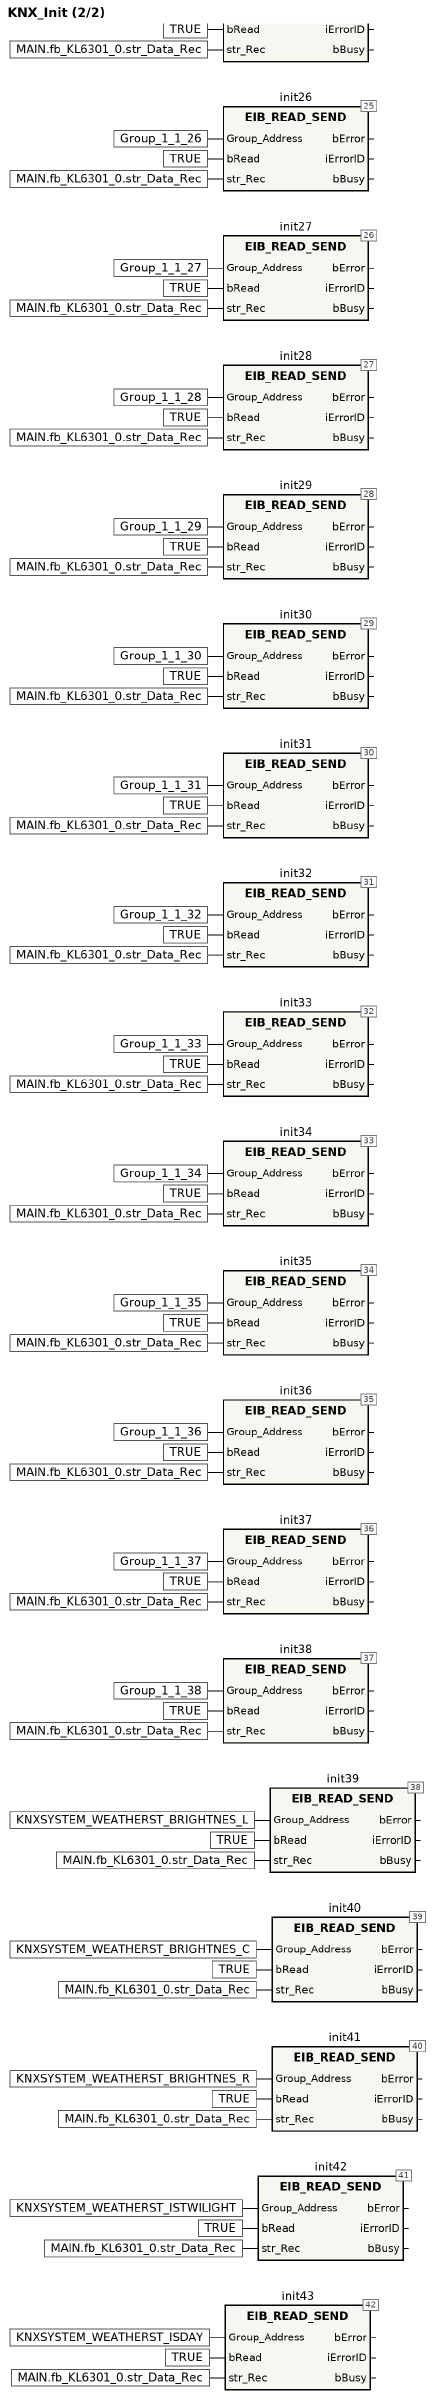
_CFC_ (* Continuous Function Chart, elements in execution order *)
#0 init1:EIB_READ_SEND(Group_Address: Group_1_1_1, bRead: TRUE, str_Rec: MAIN.fb_KL6301_0.str_Data_Rec)
#1 init2:EIB_READ_SEND(Group_Address: Group_1_1_2, bRead: TRUE, str_Rec: MAIN.fb_KL6301_0.str_Data_Rec)
#2 init3:EIB_READ_SEND(Group_Address: Group_1_1_3, bRead: TRUE, str_Rec: MAIN.fb_KL6301_0.str_Data_Rec)
#3 init4:EIB_READ_SEND(Group_Address: Group_1_1_4, bRead: TRUE, str_Rec: MAIN.fb_KL6301_0.str_Data_Rec)
#4 init5:EIB_READ_SEND(Group_Address: Group_1_1_5, bRead: TRUE, str_Rec: MAIN.fb_KL6301_0.str_Data_Rec)
#5 init6:EIB_READ_SEND(Group_Address: Group_1_1_6, bRead: TRUE, str_Rec: MAIN.fb_KL6301_0.str_Data_Rec)
#6 init7:EIB_READ_SEND(Group_Address: Group_1_1_7, bRead: TRUE, str_Rec: MAIN.fb_KL6301_0.str_Data_Rec)
#7 init8:EIB_READ_SEND(Group_Address: Group_1_1_8, bRead: TRUE, str_Rec: MAIN.fb_KL6301_0.str_Data_Rec)
#8 init9:EIB_READ_SEND(Group_Address: Group_1_1_9, bRead: TRUE, str_Rec: MAIN.fb_KL6301_0.str_Data_Rec)
#9 init10:EIB_READ_SEND(Group_Address: Group_1_1_10, bRead: TRUE, str_Rec: MAIN.fb_KL6301_0.str_Data_Rec)
#10 init11:EIB_READ_SEND(Group_Address: Group_1_1_11, bRead: TRUE, str_Rec: MAIN.fb_KL6301_0.str_Data_Rec)
#11 init12:EIB_READ_SEND(Group_Address: Group_1_1_12, bRead: TRUE, str_Rec: MAIN.fb_KL6301_0.str_Data_Rec)
#12 init13:EIB_READ_SEND(Group_Address: Group_1_1_13, bRead: TRUE, str_Rec: MAIN.fb_KL6301_0.str_Data_Rec)
#13 init14:EIB_READ_SEND(Group_Address: Group_1_1_14, bRead: TRUE, str_Rec: MAIN.fb_KL6301_0.str_Data_Rec)
#14 init15:EIB_READ_SEND(Group_Address: Group_1_1_15, bRead: TRUE, str_Rec: MAIN.fb_KL6301_0.str_Data_Rec)
#15 init16:EIB_READ_SEND(Group_Address: Group_1_1_16, bRead: TRUE, str_Rec: MAIN.fb_KL6301_0.str_Data_Rec)
#16 init17:EIB_READ_SEND(Group_Address: Group_1_1_17, bRead: TRUE, str_Rec: MAIN.fb_KL6301_0.str_Data_Rec)
#17 init18:EIB_READ_SEND(Group_Address: Group_1_1_18, bRead: TRUE, str_Rec: MAIN.fb_KL6301_0.str_Data_Rec)
#18 init19:EIB_READ_SEND(Group_Address: Group_1_1_19, bRead: TRUE, str_Rec: MAIN.fb_KL6301_0.str_Data_Rec)
#19 init20:EIB_READ_SEND(Group_Address: Group_1_1_20, bRead: TRUE, str_Rec: MAIN.fb_KL6301_0.str_Data_Rec)
#20 init21:EIB_READ_SEND(Group_Address: Group_1_1_21, bRead: TRUE, str_Rec: MAIN.fb_KL6301_0.str_Data_Rec)
#21 init22:EIB_READ_SEND(Group_Address: Group_1_1_22, bRead: TRUE, str_Rec: MAIN.fb_KL6301_0.str_Data_Rec)
#22 init23:EIB_READ_SEND(Group_Address: Group_1_1_23, bRead: TRUE, str_Rec: MAIN.fb_KL6301_0.str_Data_Rec)
#23 init24:EIB_READ_SEND(Group_Address: Group_1_1_24, bRead: TRUE, str_Rec: MAIN.fb_KL6301_0.str_Data_Rec)
#24 init25:EIB_READ_SEND(Group_Address: Group_1_1_25, bRead: TRUE, str_Rec: MAIN.fb_KL6301_0.str_Data_Rec)
#25 init26:EIB_READ_SEND(Group_Address: Group_1_1_26, bRead: TRUE, str_Rec: MAIN.fb_KL6301_0.str_Data_Rec)
#26 init27:EIB_READ_SEND(Group_Address: Group_1_1_27, bRead: TRUE, str_Rec: MAIN.fb_KL6301_0.str_Data_Rec)
#27 init28:EIB_READ_SEND(Group_Address: Group_1_1_28, bRead: TRUE, str_Rec: MAIN.fb_KL6301_0.str_Data_Rec)
#28 init29:EIB_READ_SEND(Group_Address: Group_1_1_29, bRead: TRUE, str_Rec: MAIN.fb_KL6301_0.str_Data_Rec)
#29 init30:EIB_READ_SEND(Group_Address: Group_1_1_30, bRead: TRUE, str_Rec: MAIN.fb_KL6301_0.str_Data_Rec)
#30 init31:EIB_READ_SEND(Group_Address: Group_1_1_31, bRead: TRUE, str_Rec: MAIN.fb_KL6301_0.str_Data_Rec)
#31 init32:EIB_READ_SEND(Group_Address: Group_1_1_32, bRead: TRUE, str_Rec: MAIN.fb_KL6301_0.str_Data_Rec)
#32 init33:EIB_READ_SEND(Group_Address: Group_1_1_33, bRead: TRUE, str_Rec: MAIN.fb_KL6301_0.str_Data_Rec)
#33 init34:EIB_READ_SEND(Group_Address: Group_1_1_34, bRead: TRUE, str_Rec: MAIN.fb_KL6301_0.str_Data_Rec)
#34 init35:EIB_READ_SEND(Group_Address: Group_1_1_35, bRead: TRUE, str_Rec: MAIN.fb_KL6301_0.str_Data_Rec)
#35 init36:EIB_READ_SEND(Group_Address: Group_1_1_36, bRead: TRUE, str_Rec: MAIN.fb_KL6301_0.str_Data_Rec)
#36 init37:EIB_READ_SEND(Group_Address: Group_1_1_37, bRead: TRUE, str_Rec: MAIN.fb_KL6301_0.str_Data_Rec)
#37 init38:EIB_READ_SEND(Group_Address: Group_1_1_38, bRead: TRUE, str_Rec: MAIN.fb_KL6301_0.str_Data_Rec)
#38 init39:EIB_READ_SEND(Group_Address: KNXSYSTEM_WEATHERST_BRIGHTNES_L, bRead: TRUE, str_Rec: MAIN.fb_KL6301_0.str_Data_Rec)
#39 init40:EIB_READ_SEND(Group_Address: KNXSYSTEM_WEATHERST_BRIGHTNES_C, bRead: TRUE, str_Rec: MAIN.fb_KL6301_0.str_Data_Rec)
#40 init41:EIB_READ_SEND(Group_Address: KNXSYSTEM_WEATHERST_BRIGHTNES_R, bRead: TRUE, str_Rec: MAIN.fb_KL6301_0.str_Data_Rec)
#41 init42:EIB_READ_SEND(Group_Address: KNXSYSTEM_WEATHERST_ISTWILIGHT, bRead: TRUE, str_Rec: MAIN.fb_KL6301_0.str_Data_Rec)
#42 init43:EIB_READ_SEND(Group_Address: KNXSYSTEM_WEATHERST_ISDAY, bRead: TRUE, str_Rec: MAIN.fb_KL6301_0.str_Data_Rec)
_END_CFC_
END_PROGRAM

(* POU Main_EIB_REC, CFC *)
PROGRAM Main_EIB_REC
VAR
	EIB_BIT_REC_0: EIB_BIT_REC;

(*	EIB_BIT_REC_1: EIB_BIT_REC;
	EIB_REAL_REC_0:EIB_2OCTET_FLOAT_REC;
	EIB_REAL_REC_Temp:EIB_2OCTET_FLOAT_REC;
	EIB_8Bit:EIB_8BIT_SIGN_REC;
	EIB_3Bit:EIB_3BIT_CONTROL_REC;
	EIB_3Bit_1:EIB_3BIT_CONTROL_REC;
	EIB_2BYTE_UINT:EIB_2OCTET_UNSIGN_REC;
	EIB_4UDINT:EIB_4OCTET_SIGN_REC;
	EIB_4Float:EIB_4OCTET_FLOAT_REC;  *)

	Group_1_1_1: EIB_GROUP_ADDR := (MAIN:=1,SUB_MAIN:=1,NUMBER:=1);
	Group_1_1_2: EIB_GROUP_ADDR := (MAIN:=1,SUB_MAIN:=1,NUMBER:=2);
	Group_1_1_3: EIB_GROUP_ADDR := (MAIN:=1,SUB_MAIN:=1,NUMBER:=3);
	Group_1_1_4: EIB_GROUP_ADDR := (MAIN:=1,SUB_MAIN:=1,NUMBER:=4);
	Group_1_1_5: EIB_GROUP_ADDR := (MAIN:=1,SUB_MAIN:=1,NUMBER:=5);
	Group_1_1_6: EIB_GROUP_ADDR := (MAIN:=1,SUB_MAIN:=1,NUMBER:=6);
	Group_1_1_7: EIB_GROUP_ADDR := (MAIN:=1,SUB_MAIN:=1,NUMBER:=7);
	Group_1_1_8: EIB_GROUP_ADDR := (MAIN:=1,SUB_MAIN:=1,NUMBER:=8);
	Group_1_1_9: EIB_GROUP_ADDR := (MAIN:=1,SUB_MAIN:=1,NUMBER:=9);
	Group_1_1_10: EIB_GROUP_ADDR := (MAIN:=1,SUB_MAIN:=1,NUMBER:=10);
	Group_1_1_11: EIB_GROUP_ADDR := (MAIN:=1,SUB_MAIN:=1,NUMBER:=11);
	Group_1_1_12: EIB_GROUP_ADDR := (MAIN:=1,SUB_MAIN:=1,NUMBER:=12);
	Group_1_1_13: EIB_GROUP_ADDR := (MAIN:=1,SUB_MAIN:=1,NUMBER:=13);
	Group_1_1_14: EIB_GROUP_ADDR := (MAIN:=1,SUB_MAIN:=1,NUMBER:=14);
	Group_1_1_15: EIB_GROUP_ADDR := (MAIN:=1,SUB_MAIN:=1,NUMBER:=15);
	Group_1_1_16: EIB_GROUP_ADDR := (MAIN:=1,SUB_MAIN:=1,NUMBER:=16);
	Group_1_1_17: EIB_GROUP_ADDR := (MAIN:=1,SUB_MAIN:=1,NUMBER:=17);
	Group_1_1_18: EIB_GROUP_ADDR := (MAIN:=1,SUB_MAIN:=1,NUMBER:=18);
	Group_1_1_19: EIB_GROUP_ADDR := (MAIN:=1,SUB_MAIN:=1,NUMBER:=19);
	Group_1_1_20: EIB_GROUP_ADDR := (MAIN:=1,SUB_MAIN:=1,NUMBER:=20);
	Group_1_1_21: EIB_GROUP_ADDR := (MAIN:=1,SUB_MAIN:=1,NUMBER:=21);
	Group_1_1_22: EIB_GROUP_ADDR := (MAIN:=1,SUB_MAIN:=1,NUMBER:=22);
	Group_1_1_23: EIB_GROUP_ADDR := (MAIN:=1,SUB_MAIN:=1,NUMBER:=23);
	Group_1_1_24: EIB_GROUP_ADDR := (MAIN:=1,SUB_MAIN:=1,NUMBER:=24);
	Group_1_1_25: EIB_GROUP_ADDR := (MAIN:=1,SUB_MAIN:=1,NUMBER:=25);
	Group_1_1_26: EIB_GROUP_ADDR := (MAIN:=1,SUB_MAIN:=1,NUMBER:=26);
	Group_1_1_27: EIB_GROUP_ADDR := (MAIN:=1,SUB_MAIN:=1,NUMBER:=27);
	Group_1_1_28: EIB_GROUP_ADDR := (MAIN:=1,SUB_MAIN:=1,NUMBER:=28);
	Group_1_1_29: EIB_GROUP_ADDR := (MAIN:=1,SUB_MAIN:=1,NUMBER:=29);  (*zdes bilo MAIN:=5,SUB_MAIN:=1,NUMBER:=6. Sozdal otdelnuyu peremennuyu s etim adresom nizhe*)
	Group_1_1_30: EIB_GROUP_ADDR := (MAIN:=1,SUB_MAIN:=1,NUMBER:=30);

	Group_1_1_31: EIB_GROUP_ADDR := (MAIN:=1,SUB_MAIN:=1,NUMBER:=31);
	Group_1_1_32: EIB_GROUP_ADDR := (MAIN:=1,SUB_MAIN:=1,NUMBER:=32);
	Group_1_1_33: EIB_GROUP_ADDR := (MAIN:=1,SUB_MAIN:=1,NUMBER:=33);
	Group_1_1_34: EIB_GROUP_ADDR := (MAIN:=1,SUB_MAIN:=1,NUMBER:=34);
	Group_1_1_35: EIB_GROUP_ADDR := (MAIN:=1,SUB_MAIN:=1,NUMBER:=35);
	Group_1_1_36: EIB_GROUP_ADDR := (MAIN:=1,SUB_MAIN:=1,NUMBER:=36);
	Group_1_1_37: EIB_GROUP_ADDR := (MAIN:=1,SUB_MAIN:=1,NUMBER:=37);
	Group_1_1_38: EIB_GROUP_ADDR := (MAIN:=1,SUB_MAIN:=1,NUMBER:=38);

	KNXSYSTEM_WEATHERST_BRIGHTNES_L: EIB_GROUP_ADDR := (MAIN:=5,SUB_MAIN:=1,NUMBER:=2);
	KNXSYSTEM_WEATHERST_BRIGHTNES_C: EIB_GROUP_ADDR := (MAIN:=5,SUB_MAIN:=1,NUMBER:=3);
	KNXSYSTEM_WEATHERST_BRIGHTNES_R: EIB_GROUP_ADDR := (MAIN:=5,SUB_MAIN:=1,NUMBER:=4);
	KNXSYSTEM_WEATHERST_ISTWILIGHT: EIB_GROUP_ADDR := (MAIN:=5,SUB_MAIN:=1,NUMBER:=40);
	KNXSYSTEM_WEATHERST_ISDAY: EIB_GROUP_ADDR := (MAIN:=5,SUB_MAIN:=1,NUMBER:=6);

	EIB_BIT_REC_1: EIB_BIT_REC;
	EIB_BIT_REC_2: EIB_BIT_REC;
	EIB_BIT_REC_3: EIB_BIT_REC;
	EIB_BIT_REC_4: EIB_BIT_REC;
	EIB_BIT_REC_5: EIB_BIT_REC;
	EIB_BIT_REC_6: EIB_BIT_REC;
	EIB_BIT_REC_7: EIB_BIT_REC;
	EIB_BIT_REC_8: EIB_BIT_REC;
	EIB_BIT_REC_9: EIB_BIT_REC;
	EIB_BIT_REC_10: EIB_BIT_REC;
	EIB_BIT_REC_11: EIB_BIT_REC;
	EIB_BIT_REC_12: EIB_BIT_REC;
	EIB_BIT_REC_13: EIB_BIT_REC;
	EIB_BIT_REC_14: EIB_BIT_REC;
	EIB_BIT_REC_15: EIB_BIT_REC;
	EIB_BIT_REC_16: EIB_BIT_REC;
	EIB_BIT_REC_17: EIB_BIT_REC;
	EIB_BIT_REC_18: EIB_BIT_REC;
	EIB_BIT_REC_19: EIB_BIT_REC;
	EIB_BIT_REC_20: EIB_BIT_REC;
	EIB_BIT_REC_21: EIB_BIT_REC;
	EIB_BIT_REC_22: EIB_BIT_REC;
	EIB_BIT_REC_23: EIB_BIT_REC;
	EIB_BIT_REC_24: EIB_BIT_REC;
	EIB_BIT_REC_25: EIB_BIT_REC;
	EIB_BIT_REC_26: EIB_BIT_REC;
	EIB_BIT_REC_27: EIB_BIT_REC;
	EIB_BIT_REC_28: EIB_BIT_REC;
	EIB_BIT_REC_29: EIB_BIT_REC;
	EIB_BIT_REC_30: EIB_BIT_REC;
	EIB_BIT_REC_31: EIB_BIT_REC;
	EIB_BIT_REC_32: EIB_BIT_REC;
	EIB_BIT_REC_33: EIB_BIT_REC;
	EIB_BIT_REC_34: EIB_BIT_REC;
	EIB_BIT_REC_35: EIB_BIT_REC;
	EIB_BIT_REC_36: EIB_BIT_REC;
	EIB_BIT_REC_37: EIB_BIT_REC;
	EIB_BIT_REC_38: EIB_BIT_REC;
	EIB_BIT_REC_39: EIB_BIT_REC;
	EIB_BIT_REC_40: EIB_BIT_REC;
	EIB_BIT_REC_41: EIB_BIT_REC;
	EIB_ALL_DATA_TYPES_REC_40: EIB_4OCTET_SIGN_REC;
	EIB_ALL_DATA_TYPES_REC_41: EIB_4OCTET_SIGN_REC;
	EIB_ALL_DATA_TYPES_REC_42: EIB_4OCTET_SIGN_REC;
	fb_GetTi: NT_GetTime;
	Timer1: TON;
END_VAR
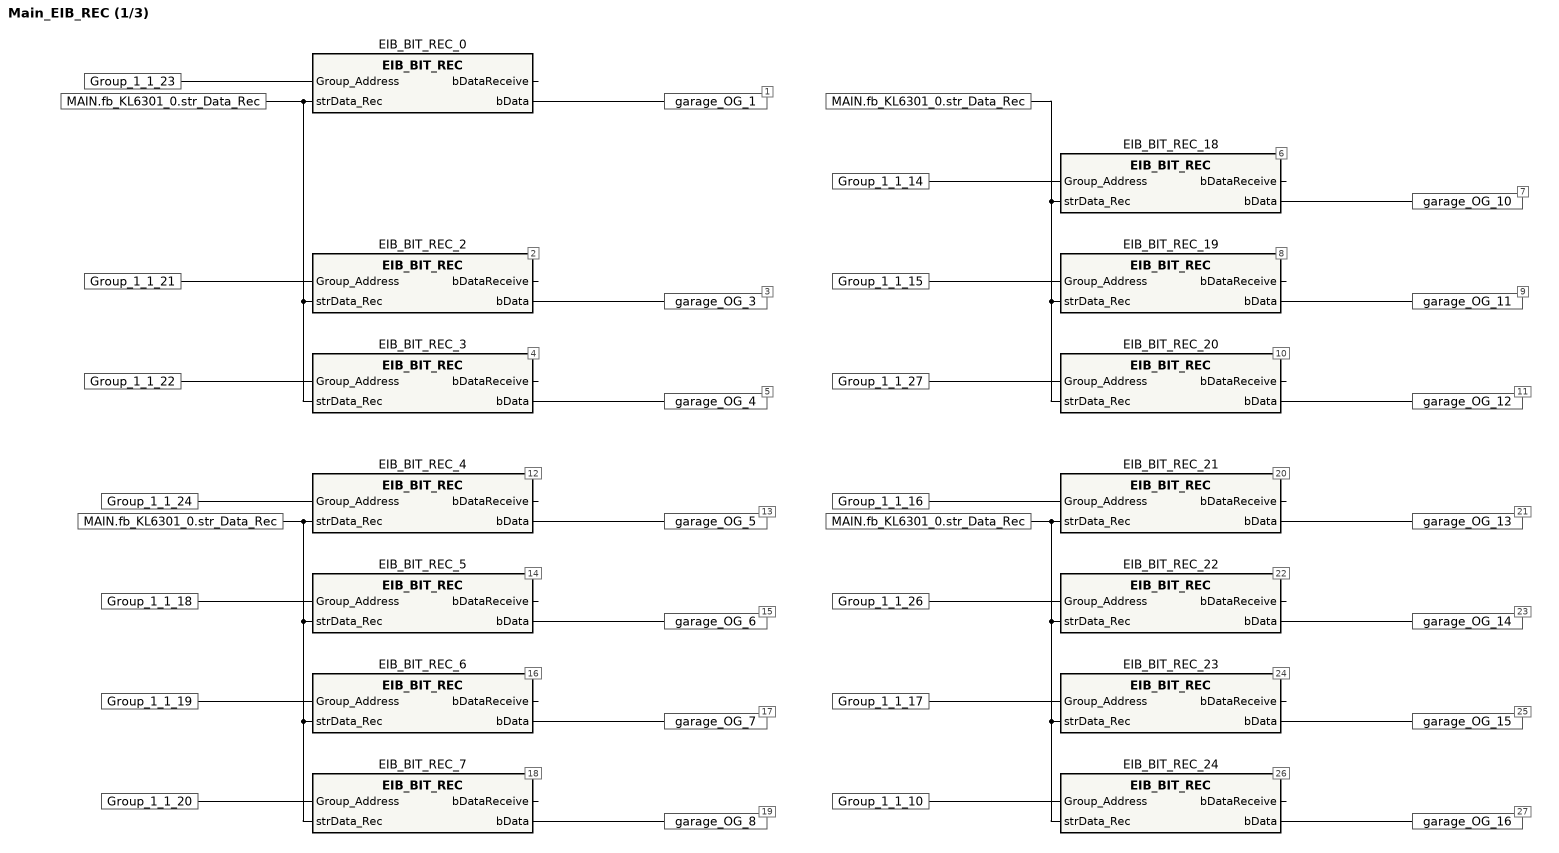
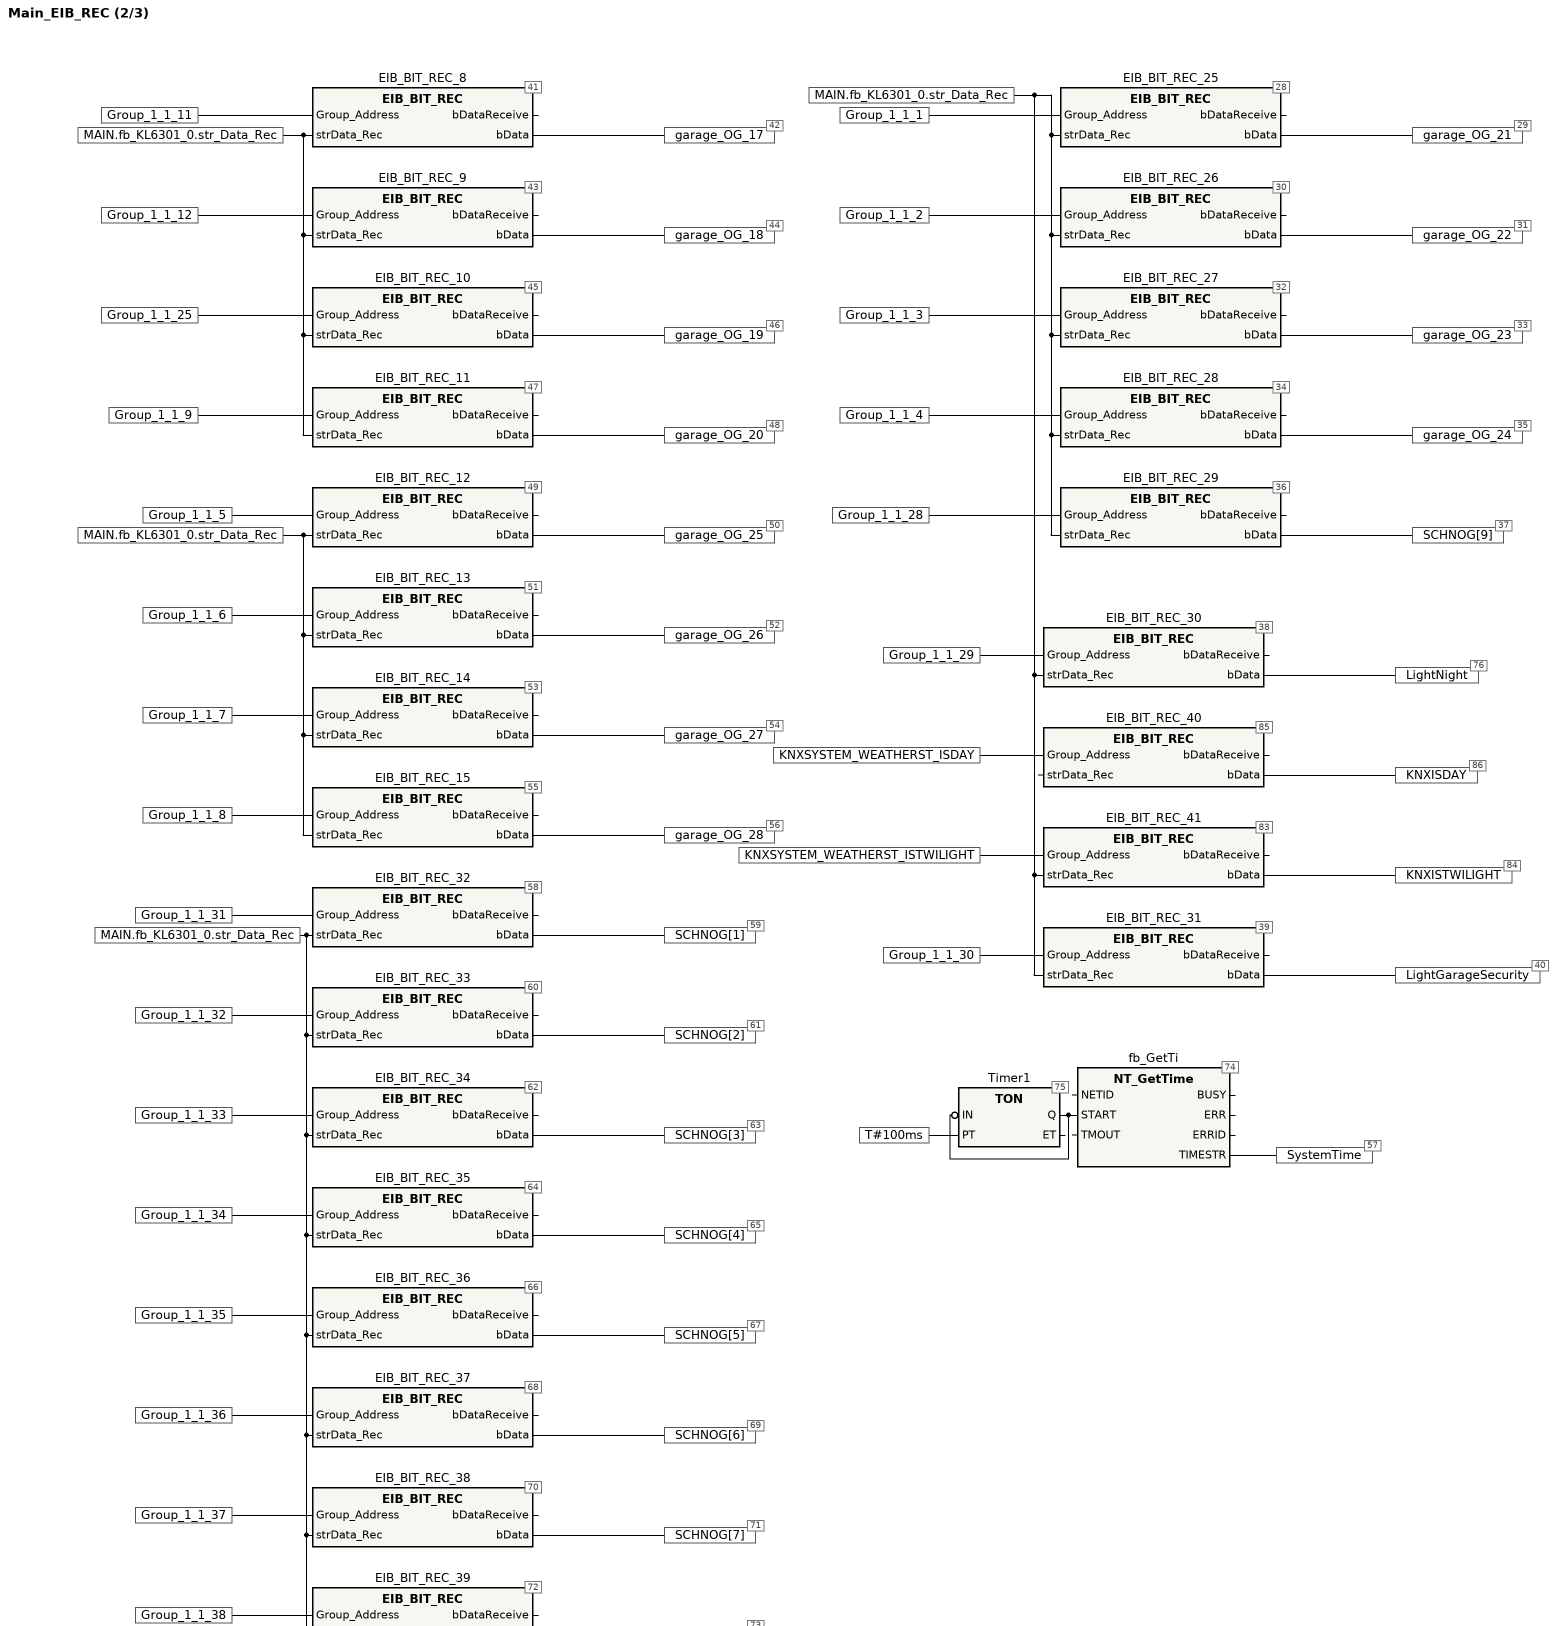
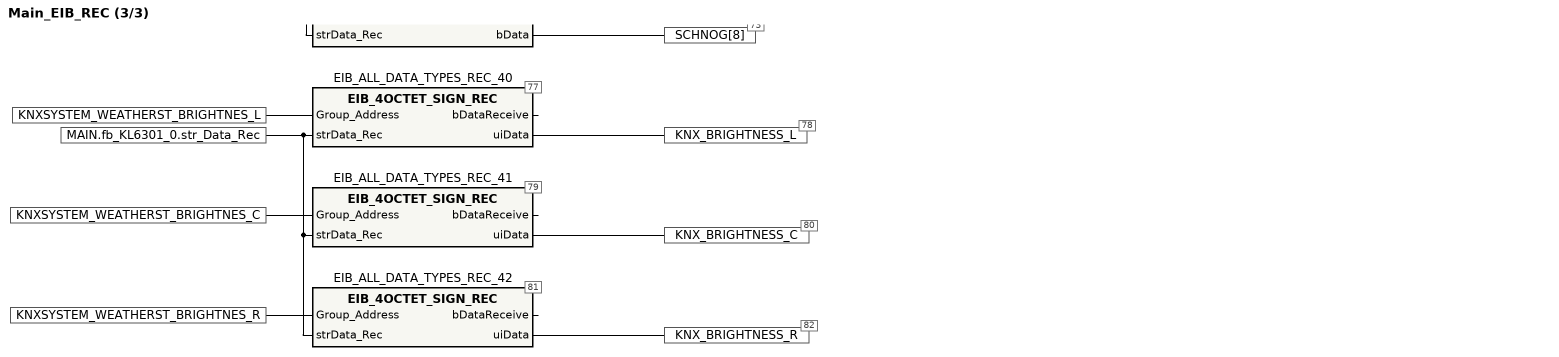
_CFC_ (* Continuous Function Chart, elements in execution order *)
#0 EIB_BIT_REC_0:EIB_BIT_REC(Group_Address: Group_1_1_23, strData_Rec: MAIN.fb_KL6301_0.str_Data_Rec)
#1 garage_OG_1 <= #0.bData
#2 EIB_BIT_REC_2:EIB_BIT_REC(Group_Address: Group_1_1_21, strData_Rec: MAIN.fb_KL6301_0.str_Data_Rec)
#3 garage_OG_3 <= #2.bData
#4 EIB_BIT_REC_3:EIB_BIT_REC(Group_Address: Group_1_1_22, strData_Rec: MAIN.fb_KL6301_0.str_Data_Rec)
#5 garage_OG_4 <= #4.bData
#6 EIB_BIT_REC_18:EIB_BIT_REC(Group_Address: Group_1_1_14, strData_Rec: MAIN.fb_KL6301_0.str_Data_Rec)
#7 garage_OG_10 <= #6.bData
#8 EIB_BIT_REC_19:EIB_BIT_REC(Group_Address: Group_1_1_15, strData_Rec: MAIN.fb_KL6301_0.str_Data_Rec)
#9 garage_OG_11 <= #8.bData
#10 EIB_BIT_REC_20:EIB_BIT_REC(Group_Address: Group_1_1_27, strData_Rec: MAIN.fb_KL6301_0.str_Data_Rec)
#11 garage_OG_12 <= #10.bData
#12 EIB_BIT_REC_4:EIB_BIT_REC(Group_Address: Group_1_1_24, strData_Rec: MAIN.fb_KL6301_0.str_Data_Rec)
#13 garage_OG_5 <= #12.bData
#14 EIB_BIT_REC_5:EIB_BIT_REC(Group_Address: Group_1_1_18, strData_Rec: MAIN.fb_KL6301_0.str_Data_Rec)
#15 garage_OG_6 <= #14.bData
#16 EIB_BIT_REC_6:EIB_BIT_REC(Group_Address: Group_1_1_19, strData_Rec: MAIN.fb_KL6301_0.str_Data_Rec)
#17 garage_OG_7 <= #16.bData
#18 EIB_BIT_REC_7:EIB_BIT_REC(Group_Address: Group_1_1_20, strData_Rec: MAIN.fb_KL6301_0.str_Data_Rec)
#19 garage_OG_8 <= #18.bData
#20 EIB_BIT_REC_21:EIB_BIT_REC(Group_Address: Group_1_1_16, strData_Rec: MAIN.fb_KL6301_0.str_Data_Rec)
#21 garage_OG_13 <= #20.bData
#22 EIB_BIT_REC_22:EIB_BIT_REC(Group_Address: Group_1_1_26, strData_Rec: MAIN.fb_KL6301_0.str_Data_Rec)
#23 garage_OG_14 <= #22.bData
#24 EIB_BIT_REC_23:EIB_BIT_REC(Group_Address: Group_1_1_17, strData_Rec: MAIN.fb_KL6301_0.str_Data_Rec)
#25 garage_OG_15 <= #24.bData
#26 EIB_BIT_REC_24:EIB_BIT_REC(Group_Address: Group_1_1_10, strData_Rec: MAIN.fb_KL6301_0.str_Data_Rec)
#27 garage_OG_16 <= #26.bData
#28 EIB_BIT_REC_25:EIB_BIT_REC(Group_Address: Group_1_1_1, strData_Rec: MAIN.fb_KL6301_0.str_Data_Rec)
#29 garage_OG_21 <= #28.bData
#30 EIB_BIT_REC_26:EIB_BIT_REC(Group_Address: Group_1_1_2, strData_Rec: MAIN.fb_KL6301_0.str_Data_Rec)
#31 garage_OG_22 <= #30.bData
#32 EIB_BIT_REC_27:EIB_BIT_REC(Group_Address: Group_1_1_3, strData_Rec: MAIN.fb_KL6301_0.str_Data_Rec)
#33 garage_OG_23 <= #32.bData
#34 EIB_BIT_REC_28:EIB_BIT_REC(Group_Address: Group_1_1_4, strData_Rec: MAIN.fb_KL6301_0.str_Data_Rec)
#35 garage_OG_24 <= #34.bData
#36 EIB_BIT_REC_29:EIB_BIT_REC(Group_Address: Group_1_1_28, strData_Rec: MAIN.fb_KL6301_0.str_Data_Rec)
#37 SCHNOG[9] <= #36.bData
#38 EIB_BIT_REC_30:EIB_BIT_REC(Group_Address: Group_1_1_29, strData_Rec: MAIN.fb_KL6301_0.str_Data_Rec)
#39 EIB_BIT_REC_31:EIB_BIT_REC(Group_Address: Group_1_1_30, strData_Rec: MAIN.fb_KL6301_0.str_Data_Rec)
#40 LightGarageSecurity <= #39.bData
#41 EIB_BIT_REC_8:EIB_BIT_REC(Group_Address: Group_1_1_11, strData_Rec: MAIN.fb_KL6301_0.str_Data_Rec)
#42 garage_OG_17 <= #41.bData
#43 EIB_BIT_REC_9:EIB_BIT_REC(Group_Address: Group_1_1_12, strData_Rec: MAIN.fb_KL6301_0.str_Data_Rec)
#44 garage_OG_18 <= #43.bData
#45 EIB_BIT_REC_10:EIB_BIT_REC(Group_Address: Group_1_1_25, strData_Rec: MAIN.fb_KL6301_0.str_Data_Rec)
#46 garage_OG_19 <= #45.bData
#47 EIB_BIT_REC_11:EIB_BIT_REC(Group_Address: Group_1_1_9, strData_Rec: MAIN.fb_KL6301_0.str_Data_Rec)
#48 garage_OG_20 <= #47.bData
#49 EIB_BIT_REC_12:EIB_BIT_REC(Group_Address: Group_1_1_5, strData_Rec: MAIN.fb_KL6301_0.str_Data_Rec)
#50 garage_OG_25 <= #49.bData
#51 EIB_BIT_REC_13:EIB_BIT_REC(Group_Address: Group_1_1_6, strData_Rec: MAIN.fb_KL6301_0.str_Data_Rec)
#52 garage_OG_26 <= #51.bData
#53 EIB_BIT_REC_14:EIB_BIT_REC(Group_Address: Group_1_1_7, strData_Rec: MAIN.fb_KL6301_0.str_Data_Rec)
#54 garage_OG_27 <= #53.bData
#55 EIB_BIT_REC_15:EIB_BIT_REC(Group_Address: Group_1_1_8, strData_Rec: MAIN.fb_KL6301_0.str_Data_Rec)
#56 garage_OG_28 <= #55.bData
#57 SystemTime <= #74.TIMESTR
#58 EIB_BIT_REC_32:EIB_BIT_REC(Group_Address: Group_1_1_31, strData_Rec: MAIN.fb_KL6301_0.str_Data_Rec)
#59 SCHNOG[1] <= #58.bData
#60 EIB_BIT_REC_33:EIB_BIT_REC(Group_Address: Group_1_1_32, strData_Rec: MAIN.fb_KL6301_0.str_Data_Rec)
#61 SCHNOG[2] <= #60.bData
#62 EIB_BIT_REC_34:EIB_BIT_REC(Group_Address: Group_1_1_33, strData_Rec: MAIN.fb_KL6301_0.str_Data_Rec)
#63 SCHNOG[3] <= #62.bData
#64 EIB_BIT_REC_35:EIB_BIT_REC(Group_Address: Group_1_1_34, strData_Rec: MAIN.fb_KL6301_0.str_Data_Rec)
#65 SCHNOG[4] <= #64.bData
#66 EIB_BIT_REC_36:EIB_BIT_REC(Group_Address: Group_1_1_35, strData_Rec: MAIN.fb_KL6301_0.str_Data_Rec)
#67 SCHNOG[5] <= #66.bData
#68 EIB_BIT_REC_37:EIB_BIT_REC(Group_Address: Group_1_1_36, strData_Rec: MAIN.fb_KL6301_0.str_Data_Rec)
#69 SCHNOG[6] <= #68.bData
#70 EIB_BIT_REC_38:EIB_BIT_REC(Group_Address: Group_1_1_37, strData_Rec: MAIN.fb_KL6301_0.str_Data_Rec)
#71 SCHNOG[7] <= #70.bData
#72 EIB_BIT_REC_39:EIB_BIT_REC(Group_Address: Group_1_1_38, strData_Rec: MAIN.fb_KL6301_0.str_Data_Rec)
#73 SCHNOG[8] <= #72.bData
#74 fb_GetTi:NT_GetTime(NETID: -, START: #75.Q, TMOUT: -)
#75 Timer1:TON(IN: NOT #75.Q, PT: T#100ms)
#76 LightNight <= #38.bData
#77 EIB_ALL_DATA_TYPES_REC_40:EIB_4OCTET_SIGN_REC(Group_Address: KNXSYSTEM_WEATHERST_BRIGHTNES_L, strData_Rec: MAIN.fb_KL6301_0.str_Data_Rec)
#78 KNX_BRIGHTNESS_L <= #77.uiData
#79 EIB_ALL_DATA_TYPES_REC_41:EIB_4OCTET_SIGN_REC(Group_Address: KNXSYSTEM_WEATHERST_BRIGHTNES_C, strData_Rec: MAIN.fb_KL6301_0.str_Data_Rec)
#80 KNX_BRIGHTNESS_C <= #79.uiData
#81 EIB_ALL_DATA_TYPES_REC_42:EIB_4OCTET_SIGN_REC(Group_Address: KNXSYSTEM_WEATHERST_BRIGHTNES_R, strData_Rec: MAIN.fb_KL6301_0.str_Data_Rec)
#82 KNX_BRIGHTNESS_R <= #81.uiData
#83 EIB_BIT_REC_41:EIB_BIT_REC(Group_Address: KNXSYSTEM_WEATHERST_ISTWILIGHT, strData_Rec: MAIN.fb_KL6301_0.str_Data_Rec)
#84 KNXISTWILIGHT <= #83.bData
#85 EIB_BIT_REC_40:EIB_BIT_REC(Group_Address: KNXSYSTEM_WEATHERST_ISDAY, strData_Rec: -)
#86 KNXISDAY <= #85.bData
_END_CFC_
(* the same logic as Structured Text *)
EIB_BIT_REC_0(Group_Address := Group_1_1_23, strData_Rec := MAIN.fb_KL6301_0.str_Data_Rec);
garage_OG_1 := EIB_BIT_REC_0.bData;
EIB_BIT_REC_2(Group_Address := Group_1_1_21, strData_Rec := MAIN.fb_KL6301_0.str_Data_Rec);
garage_OG_3 := EIB_BIT_REC_2.bData;
EIB_BIT_REC_3(Group_Address := Group_1_1_22, strData_Rec := MAIN.fb_KL6301_0.str_Data_Rec);
garage_OG_4 := EIB_BIT_REC_3.bData;
EIB_BIT_REC_18(Group_Address := Group_1_1_14, strData_Rec := MAIN.fb_KL6301_0.str_Data_Rec);
garage_OG_10 := EIB_BIT_REC_18.bData;
EIB_BIT_REC_19(Group_Address := Group_1_1_15, strData_Rec := MAIN.fb_KL6301_0.str_Data_Rec);
garage_OG_11 := EIB_BIT_REC_19.bData;
EIB_BIT_REC_20(Group_Address := Group_1_1_27, strData_Rec := MAIN.fb_KL6301_0.str_Data_Rec);
garage_OG_12 := EIB_BIT_REC_20.bData;
EIB_BIT_REC_4(Group_Address := Group_1_1_24, strData_Rec := MAIN.fb_KL6301_0.str_Data_Rec);
garage_OG_5 := EIB_BIT_REC_4.bData;
EIB_BIT_REC_5(Group_Address := Group_1_1_18, strData_Rec := MAIN.fb_KL6301_0.str_Data_Rec);
garage_OG_6 := EIB_BIT_REC_5.bData;
EIB_BIT_REC_6(Group_Address := Group_1_1_19, strData_Rec := MAIN.fb_KL6301_0.str_Data_Rec);
garage_OG_7 := EIB_BIT_REC_6.bData;
EIB_BIT_REC_7(Group_Address := Group_1_1_20, strData_Rec := MAIN.fb_KL6301_0.str_Data_Rec);
garage_OG_8 := EIB_BIT_REC_7.bData;
EIB_BIT_REC_21(Group_Address := Group_1_1_16, strData_Rec := MAIN.fb_KL6301_0.str_Data_Rec);
garage_OG_13 := EIB_BIT_REC_21.bData;
EIB_BIT_REC_22(Group_Address := Group_1_1_26, strData_Rec := MAIN.fb_KL6301_0.str_Data_Rec);
garage_OG_14 := EIB_BIT_REC_22.bData;
EIB_BIT_REC_23(Group_Address := Group_1_1_17, strData_Rec := MAIN.fb_KL6301_0.str_Data_Rec);
garage_OG_15 := EIB_BIT_REC_23.bData;
EIB_BIT_REC_24(Group_Address := Group_1_1_10, strData_Rec := MAIN.fb_KL6301_0.str_Data_Rec);
garage_OG_16 := EIB_BIT_REC_24.bData;
EIB_BIT_REC_25(Group_Address := Group_1_1_1, strData_Rec := MAIN.fb_KL6301_0.str_Data_Rec);
garage_OG_21 := EIB_BIT_REC_25.bData;
EIB_BIT_REC_26(Group_Address := Group_1_1_2, strData_Rec := MAIN.fb_KL6301_0.str_Data_Rec);
garage_OG_22 := EIB_BIT_REC_26.bData;
EIB_BIT_REC_27(Group_Address := Group_1_1_3, strData_Rec := MAIN.fb_KL6301_0.str_Data_Rec);
garage_OG_23 := EIB_BIT_REC_27.bData;
EIB_BIT_REC_28(Group_Address := Group_1_1_4, strData_Rec := MAIN.fb_KL6301_0.str_Data_Rec);
garage_OG_24 := EIB_BIT_REC_28.bData;
EIB_BIT_REC_29(Group_Address := Group_1_1_28, strData_Rec := MAIN.fb_KL6301_0.str_Data_Rec);
SCHNOG[9] := EIB_BIT_REC_29.bData;
EIB_BIT_REC_30(Group_Address := Group_1_1_29, strData_Rec := MAIN.fb_KL6301_0.str_Data_Rec);
EIB_BIT_REC_31(Group_Address := Group_1_1_30, strData_Rec := MAIN.fb_KL6301_0.str_Data_Rec);
LightGarageSecurity := EIB_BIT_REC_31.bData;
EIB_BIT_REC_8(Group_Address := Group_1_1_11, strData_Rec := MAIN.fb_KL6301_0.str_Data_Rec);
garage_OG_17 := EIB_BIT_REC_8.bData;
EIB_BIT_REC_9(Group_Address := Group_1_1_12, strData_Rec := MAIN.fb_KL6301_0.str_Data_Rec);
garage_OG_18 := EIB_BIT_REC_9.bData;
EIB_BIT_REC_10(Group_Address := Group_1_1_25, strData_Rec := MAIN.fb_KL6301_0.str_Data_Rec);
garage_OG_19 := EIB_BIT_REC_10.bData;
EIB_BIT_REC_11(Group_Address := Group_1_1_9, strData_Rec := MAIN.fb_KL6301_0.str_Data_Rec);
garage_OG_20 := EIB_BIT_REC_11.bData;
EIB_BIT_REC_12(Group_Address := Group_1_1_5, strData_Rec := MAIN.fb_KL6301_0.str_Data_Rec);
garage_OG_25 := EIB_BIT_REC_12.bData;
EIB_BIT_REC_13(Group_Address := Group_1_1_6, strData_Rec := MAIN.fb_KL6301_0.str_Data_Rec);
garage_OG_26 := EIB_BIT_REC_13.bData;
EIB_BIT_REC_14(Group_Address := Group_1_1_7, strData_Rec := MAIN.fb_KL6301_0.str_Data_Rec);
garage_OG_27 := EIB_BIT_REC_14.bData;
EIB_BIT_REC_15(Group_Address := Group_1_1_8, strData_Rec := MAIN.fb_KL6301_0.str_Data_Rec);
garage_OG_28 := EIB_BIT_REC_15.bData;
SystemTime := fb_GetTi.TIMESTR;
EIB_BIT_REC_32(Group_Address := Group_1_1_31, strData_Rec := MAIN.fb_KL6301_0.str_Data_Rec);
SCHNOG[1] := EIB_BIT_REC_32.bData;
EIB_BIT_REC_33(Group_Address := Group_1_1_32, strData_Rec := MAIN.fb_KL6301_0.str_Data_Rec);
SCHNOG[2] := EIB_BIT_REC_33.bData;
EIB_BIT_REC_34(Group_Address := Group_1_1_33, strData_Rec := MAIN.fb_KL6301_0.str_Data_Rec);
SCHNOG[3] := EIB_BIT_REC_34.bData;
EIB_BIT_REC_35(Group_Address := Group_1_1_34, strData_Rec := MAIN.fb_KL6301_0.str_Data_Rec);
SCHNOG[4] := EIB_BIT_REC_35.bData;
EIB_BIT_REC_36(Group_Address := Group_1_1_35, strData_Rec := MAIN.fb_KL6301_0.str_Data_Rec);
SCHNOG[5] := EIB_BIT_REC_36.bData;
EIB_BIT_REC_37(Group_Address := Group_1_1_36, strData_Rec := MAIN.fb_KL6301_0.str_Data_Rec);
SCHNOG[6] := EIB_BIT_REC_37.bData;
EIB_BIT_REC_38(Group_Address := Group_1_1_37, strData_Rec := MAIN.fb_KL6301_0.str_Data_Rec);
SCHNOG[7] := EIB_BIT_REC_38.bData;
EIB_BIT_REC_39(Group_Address := Group_1_1_38, strData_Rec := MAIN.fb_KL6301_0.str_Data_Rec);
SCHNOG[8] := EIB_BIT_REC_39.bData;
fb_GetTi(START := Timer1.Q);
Timer1(IN := NOT Timer1.Q, PT := T#100ms);
LightNight := EIB_BIT_REC_30.bData;
EIB_ALL_DATA_TYPES_REC_40(Group_Address := KNXSYSTEM_WEATHERST_BRIGHTNES_L, strData_Rec := MAIN.fb_KL6301_0.str_Data_Rec);
KNX_BRIGHTNESS_L := EIB_ALL_DATA_TYPES_REC_40.uiData;
EIB_ALL_DATA_TYPES_REC_41(Group_Address := KNXSYSTEM_WEATHERST_BRIGHTNES_C, strData_Rec := MAIN.fb_KL6301_0.str_Data_Rec);
KNX_BRIGHTNESS_C := EIB_ALL_DATA_TYPES_REC_41.uiData;
EIB_ALL_DATA_TYPES_REC_42(Group_Address := KNXSYSTEM_WEATHERST_BRIGHTNES_R, strData_Rec := MAIN.fb_KL6301_0.str_Data_Rec);
KNX_BRIGHTNESS_R := EIB_ALL_DATA_TYPES_REC_42.uiData;
EIB_BIT_REC_41(Group_Address := KNXSYSTEM_WEATHERST_ISTWILIGHT, strData_Rec := MAIN.fb_KL6301_0.str_Data_Rec);
KNXISTWILIGHT := EIB_BIT_REC_41.bData;
EIB_BIT_REC_40(Group_Address := KNXSYSTEM_WEATHERST_ISDAY);
KNXISDAY := EIB_BIT_REC_40.bData;
END_PROGRAM

(* POU POWER_OFF_TEST, ST *)
(*
power switch off priority

km name			priority
7 - schrov		1		first to switch off
3 - parouvl		2
1 - schavp1		3
9 - schuf			4
4 - schnvd		5
5 - schrb			6
10 - schno		7
11 - hammam		8
6 - schl			9
8 - schss			10
2 - schrd			11  last to switch off
*)
PROGRAM POWER_OFF_TEST
VAR
	init: INT := 0;
	test_power: REAL:=20.0;
	test_power_new: REAL:=50;
	test_power_first: REAL := 58;

	time_limit: REAL := 1;
	my_time: REAL := 0;


	flag: BOOL := FALSE;
	start: BOOL:=FALSE;

	(*Central function. All Off Garage*)
	Group_3_1_0: EIB_GROUP_ADDR := (MAIN:=3,SUB_MAIN:=1,NUMBER:=0);
	Group_3_1_1: EIB_GROUP_ADDR := (MAIN:=3,SUB_MAIN:=1,NUMBER:=1);
	Group_3_1_2: EIB_GROUP_ADDR := (MAIN:=3,SUB_MAIN:=1,NUMBER:=2);
	Group_3_1_3: EIB_GROUP_ADDR := (MAIN:=3,SUB_MAIN:=1,NUMBER:=3);
	Group_3_1_4: EIB_GROUP_ADDR := (MAIN:=3,SUB_MAIN:=1,NUMBER:=4);
	Group_3_1_5: EIB_GROUP_ADDR := (MAIN:=3,SUB_MAIN:=1,NUMBER:=5);
	Group_3_1_6: EIB_GROUP_ADDR := (MAIN:=3,SUB_MAIN:=1,NUMBER:=6);
	Group_3_1_7: EIB_GROUP_ADDR := (MAIN:=3,SUB_MAIN:=1,NUMBER:=7);
	Group_3_1_8: EIB_GROUP_ADDR := (MAIN:=3,SUB_MAIN:=1,NUMBER:=8);
	Group_3_1_9: EIB_GROUP_ADDR := (MAIN:=3,SUB_MAIN:=1,NUMBER:=9);
	Group_3_1_10: EIB_GROUP_ADDR := (MAIN:=3,SUB_MAIN:=1,NUMBER:=10);
	Group_3_1_11: EIB_GROUP_ADDR := (MAIN:=3,SUB_MAIN:=1,NUMBER:=11);

	EIB_SEND1: EIB_BIT_SEND;
	EIB_SEND2: EIB_BIT_SEND;
	EIB_SEND3: EIB_BIT_SEND;
	EIB_SEND4: EIB_BIT_SEND;
	EIB_SEND5: EIB_BIT_SEND;
	EIB_SEND6: EIB_BIT_SEND;
	EIB_SEND7: EIB_BIT_SEND;
	EIB_SEND8: EIB_BIT_SEND;
	EIB_SEND9: EIB_BIT_SEND;
	EIB_SEND10: EIB_BIT_SEND;
	EIB_SEND11: EIB_BIT_SEND;

	counter: INT := 0;
END_VAR
(***********************)
(*system testing*)
(*************************)
(*
	IF start=TRUE THEN
		test_power := test_power_first;
		flag:=TRUE;
		start:=FALSE;
	END_IF;
*)

test_power := KL3403_2_P;

CASE init OF

(*init of constants*)
0:
	power_VRU_value[1]  := 9.2;				(*km 1.7*)
	power_VRU_value[2]  := 26.25;			(*km 1.3*)
	power_VRU_value[3]  := 27.7;			(*km 1.1*)
	power_VRU_value[4]  := 1.56;			(*km 1.9*)
	power_VRU_value[5]  := 14.0;			(*km 1.4*)
	power_VRU_value[6]  := 9.1;				(*km 1.5*)
	power_VRU_value[7]  := 0;  (*29.5*)		(*km 1.10*)
	power_VRU_value[8]  := 9.0;				(*km 1.11*)
	power_VRU_value[9]  := 7.2;				(*km 1.6*)
	power_VRU_value[10]  := 9.5;			(*km 1.8*)
	power_VRU_value[11]  := 65.2;			(*km 1.2*)

	power_VRU_address[1] := Group_3_1_7;
	power_VRU_address[2] := Group_3_1_3;
	power_VRU_address[3] := Group_3_1_1;
	power_VRU_address[4] := Group_3_1_9;
	power_VRU_address[5] := Group_3_1_4;
	power_VRU_address[6] := Group_3_1_5;
	power_VRU_address[7] := Group_3_1_10;
	power_VRU_address[8] := Group_3_1_11;
	power_VRU_address[9] := Group_3_1_6;
	power_VRU_address[10] := Group_3_1_8;
	power_VRU_address[11] := Group_3_1_2;


	Current_switch_pos := 0;
	POWER_LIMIT := 55.0;

	counter := 1;

	WHILE counter <= 11 DO
		power_VRU_switch[counter] := TRUE;
		counter:=counter+1;
	END_WHILE;

	init := 1;

1:

	IF(test_power > POWER_LIMIT) THEN
(*switch off  *)
		IF(current_switch_pos < 10) THEN
			current_switch_pos := current_switch_pos + 1;
		ELSIF (test_power > power_VRU_value[11] ) THEN
			current_switch_pos := 11;
		END_IF;
	ELSE
(*switch on  *)
		IF((current_switch_pos <= 11) AND (current_switch_pos > 0)) THEN
			IF((test_power + power_VRU_value[current_switch_pos]) < POWER_LIMIT) THEN
				current_switch_pos:=current_switch_pos-1;
			END_IF;
		END_IF;
	END_IF;

	counter := 1;

	WHILE counter <= 11 DO

		IF(counter <= current_switch_pos) THEN
			power_VRU_switch[counter] := FALSE;
		ELSE
			power_VRU_switch[counter] := TRUE;
		END_IF;

		counter:=counter+1;
	END_WHILE;

(*

	IF FLAG=TRUE THEN
		IF test_power > 55 THEN
			IF(my_time > time_limit) THEN
				test_power := test_power_new;
				flag:=FALSE;
			END_IF;
		END_IF;

	my_time := my_time + 1;
	END_IF;
*)
END_CASE;

IF PowerSystemSwitcher = TRUE THEN

EIB_SEND1(Group_Address:= power_VRU_address[1], bData :=power_VRU_switch[1], str_Rec :=MAIN.fb_KL6301_0.str_Data_Rec);
EIB_SEND2(Group_Address:= power_VRU_address[2], bData :=power_VRU_switch[2], str_Rec :=MAIN.fb_KL6301_0.str_Data_Rec);
EIB_SEND3(Group_Address:= power_VRU_address[3], bData :=power_VRU_switch[3], str_Rec :=MAIN.fb_KL6301_0.str_Data_Rec);
EIB_SEND4(Group_Address:= power_VRU_address[4], bData :=power_VRU_switch[4], str_Rec :=MAIN.fb_KL6301_0.str_Data_Rec);
EIB_SEND5(Group_Address:= power_VRU_address[5], bData :=power_VRU_switch[5], str_Rec :=MAIN.fb_KL6301_0.str_Data_Rec);
EIB_SEND6(Group_Address:= power_VRU_address[6], bData :=power_VRU_switch[6], str_Rec :=MAIN.fb_KL6301_0.str_Data_Rec);
EIB_SEND7(Group_Address:= power_VRU_address[7], bData :=power_VRU_switch[7], str_Rec :=MAIN.fb_KL6301_0.str_Data_Rec);
EIB_SEND8(Group_Address:= power_VRU_address[8], bData :=power_VRU_switch[8], str_Rec :=MAIN.fb_KL6301_0.str_Data_Rec);
EIB_SEND9(Group_Address:= power_VRU_address[9], bData :=power_VRU_switch[9], str_Rec :=MAIN.fb_KL6301_0.str_Data_Rec);
EIB_SEND10(Group_Address:= power_VRU_address[10], bData :=power_VRU_switch[10], str_Rec :=MAIN.fb_KL6301_0.str_Data_Rec);
EIB_SEND11(Group_Address:= power_VRU_address[11], bData :=power_VRU_switch[11], str_Rec :=MAIN.fb_KL6301_0.str_Data_Rec);

END_IF;
END_PROGRAM

(* POU Udp_send_packet_init, ST *)
PROGRAM Udp_send_packet_init
VAR
	i: INT := 1;
	j: INT := 1;
	k: INT := 1;
	l: INT := 1;
END_VAR
Main_udp_packet.title_packet_code := 1;
Main_udp_packet.grsch_P[1] := REAL_TO_INT(KL3403_1_P * 1000);
Main_udp_packet.grsch_P[2] := REAL_TO_INT(KL3403_2_P * 1000);
Main_udp_packet.grsch_P[3] := REAL_TO_INT(KL3403_3_P * 1000);
Main_udp_packet.grsch_P[4] := REAL_TO_INT(KL3403_4_P * 1000);
Main_udp_packet.grsch_P[5] := REAL_TO_INT(KL3403_5_P * 1000);
Main_udp_packet.grsch_V[1] := REAL_TO_INT(KL3403_1_V * 1000);
Main_udp_packet.grsch_V[2] := REAL_TO_INT(KL3403_2_V * 1000);
Main_udp_packet.grsch_V[3] := REAL_TO_INT(KL3403_3_V * 1000);
Main_udp_packet.grsch_V[4] := REAL_TO_INT(KL3403_4_V * 1000);
Main_udp_packet.grsch_V[5] := REAL_TO_INT(KL3403_5_V * 1000);
Main_udp_packet.grsch_I[1] := REAL_TO_INT(KL3403_1_I * 1000);
Main_udp_packet.grsch_I[2] := REAL_TO_INT(KL3403_2_I * 1000);
Main_udp_packet.grsch_I[3] := REAL_TO_INT(KL3403_3_I * 1000);
Main_udp_packet.grsch_I[4] := REAL_TO_INT(KL3403_4_I * 1000);
Main_udp_packet.grsch_I[5] := REAL_TO_INT(KL3403_5_I * 1000);
Main_udp_packet.grsch_garage_og[1]   := BOOL_TO_INT(garage_OG_1);
Main_udp_packet.grsch_garage_og[2]   := BOOL_TO_INT(garage_OG_2);
Main_udp_packet.grsch_garage_og[3]   := BOOL_TO_INT(garage_OG_3);
Main_udp_packet.grsch_garage_og[4]   := BOOL_TO_INT(garage_OG_4);
Main_udp_packet.grsch_garage_og[5]   := BOOL_TO_INT(garage_OG_5);
Main_udp_packet.grsch_garage_og[6]   := BOOL_TO_INT(garage_OG_6);
Main_udp_packet.grsch_garage_og[7]   := BOOL_TO_INT(garage_OG_7);
Main_udp_packet.grsch_garage_og[8]   := BOOL_TO_INT(garage_OG_8);
Main_udp_packet.grsch_garage_og[9]   := BOOL_TO_INT(garage_OG_9);
Main_udp_packet.grsch_garage_og[10] := BOOL_TO_INT(garage_OG_10);
Main_udp_packet.grsch_garage_og[11] := BOOL_TO_INT(garage_OG_11);
Main_udp_packet.grsch_garage_og[12] := BOOL_TO_INT(garage_OG_12);
Main_udp_packet.grsch_garage_og[13] := BOOL_TO_INT(garage_OG_13);
Main_udp_packet.grsch_garage_og[14] := BOOL_TO_INT(garage_OG_14);
Main_udp_packet.grsch_garage_og[15] := BOOL_TO_INT(garage_OG_15);
Main_udp_packet.grsch_garage_og[16] := BOOL_TO_INT(garage_OG_16);
Main_udp_packet.grsch_garage_og[17] := BOOL_TO_INT(garage_OG_17);
Main_udp_packet.grsch_garage_og[18] := BOOL_TO_INT(garage_OG_18);
Main_udp_packet.grsch_garage_og[19] := BOOL_TO_INT(garage_OG_19);
Main_udp_packet.grsch_garage_og[20] := BOOL_TO_INT(garage_OG_20);
Main_udp_packet.grsch_garage_og[21] := BOOL_TO_INT(garage_OG_21);
Main_udp_packet.grsch_garage_og[22] := BOOL_TO_INT(garage_OG_22);
Main_udp_packet.grsch_garage_og[23] := BOOL_TO_INT(garage_OG_23);
Main_udp_packet.grsch_garage_og[24] := BOOL_TO_INT(garage_OG_24);
Main_udp_packet.grsch_garage_og[25] := BOOL_TO_INT(garage_OG_25);
Main_udp_packet.grsch_garage_og[26] := BOOL_TO_INT(garage_OG_26);
Main_udp_packet.grsch_garage_og[27] := BOOL_TO_INT(garage_OG_27);
Main_udp_packet.grsch_garage_og[28] := BOOL_TO_INT(garage_OG_28);
Main_udp_packet.grsch_garage_og[29] := BOOL_TO_INT(garage_OG_29);
FOR i := 1 TO 11 DO
Main_udp_packet.grsch_power_VRU_value[i] := REAL_TO_INT(power_VRU_value[i] * 1000);
END_FOR;
FOR j := 1 TO 11 DO
Main_udp_packet.grsch_power_VRU_switch[i] := BOOL_TO_INT(power_VRU_switch[i]);
END_FOR;
Main_udp_packet.grsch_power_limit := REAL_TO_INT(Power_limit * 1000);
Main_udp_packet.grsch_current_switch_pos := Current_switch_pos;
Main_udp_packet.grsch_SHUF_PRESSED := BOOL_TO_INT(SHUF_PRESSED);
Main_udp_packet.grsch_power_system_switcher := BOOL_TO_INT(PowerSystemSwitcher);

Main_udp_packet.schav_stack := schav_receive_stack;
FOR k := 1 TO 19 DO
Main_udp_packet.schnog_stack[k] := BOOL_TO_INT(schnog_receive_stack[k]);
END_FOR;
FOR l := 1 TO 116 DO
Main_udp_packet.schszp_stack[l] := BOOL_TO_INT(schszp_receive_stack[l]);
END_FOR;
Fletcher_checksum;
Main_udp_packet.title_packet_crc := Checksum_send;

IF (schszp_receive_stack[65] = FALSE AND schszp_force_stack[66] = TRUE) THEN schszp_force_stack[66] := FALSE; END_IF;
END_PROGRAM

(* POU Fletcher_checksum, ST *)
PROGRAM Fletcher_checksum
VAR
	Data_massive1 AT %MB756: ARRAY[1..4] OF BYTE;
	Data_massive2 AT %MB2006: ARRAY[1..424] OF BYTE;
	i: INT;
	j: INT;
	Sum1: INT;
	Sum2: INT;
	Sum3: INT;
	Sum4: INT;
END_VAR
Checksum_send := 0;
Checksum_incom := 0;
i := 0;
j := 0;
Sum1 := 0;
Sum2 := 0;
Sum3 := 0;
Sum4 := 0;

FOR i := 1 TO (PacketSize) DO
Sum1 := (Sum1 + Data_massive1[i]) MOD 255;
Sum2 := (Sum1 + Sum2) MOD 255;
END_FOR;
Checksum_incom := SHL(Sum2, 8) + Sum1;

FOR j := 1 TO (424) DO
Sum3 := (Sum3 + Data_massive2[j]) MOD 255;
Sum4 := (Sum3 + Sum4) MOD 255;
END_FOR;
Checksum_send := SHL(Sum4, 8) + Sum3;
END_PROGRAM

(* POU PeerToPeer, CFC *)
PROGRAM PeerToPeer
VAR
	rHOST_IP : STRING(15) := '192.168.3.204';
	rHOST_port : UDINT := 49161;
	lHOST_port : UDINT := 49187;
	fbSockClAll: FB_SocketCloseAll;
	fbSockUdpCr: FB_SocketUdpCreate;
	UdpSocket: T_HSocket;
	fbSockUdpRecFr: FB_SocketUdpReceiveFrom;
	fbSockUdpST: FB_SocketUdpSendTo;
	fbSockUdpSTConf: FB_SocketUdpSendTo;

	Timer1: TON;
	Timer2: TON;
	HandleString : STRING(80);
	Timer3: TON;
END_VAR
VAR (* helpers for the ST form of the networks *)
	_t29 : BOOL;
	_t76 : BOOL;
END_VAR
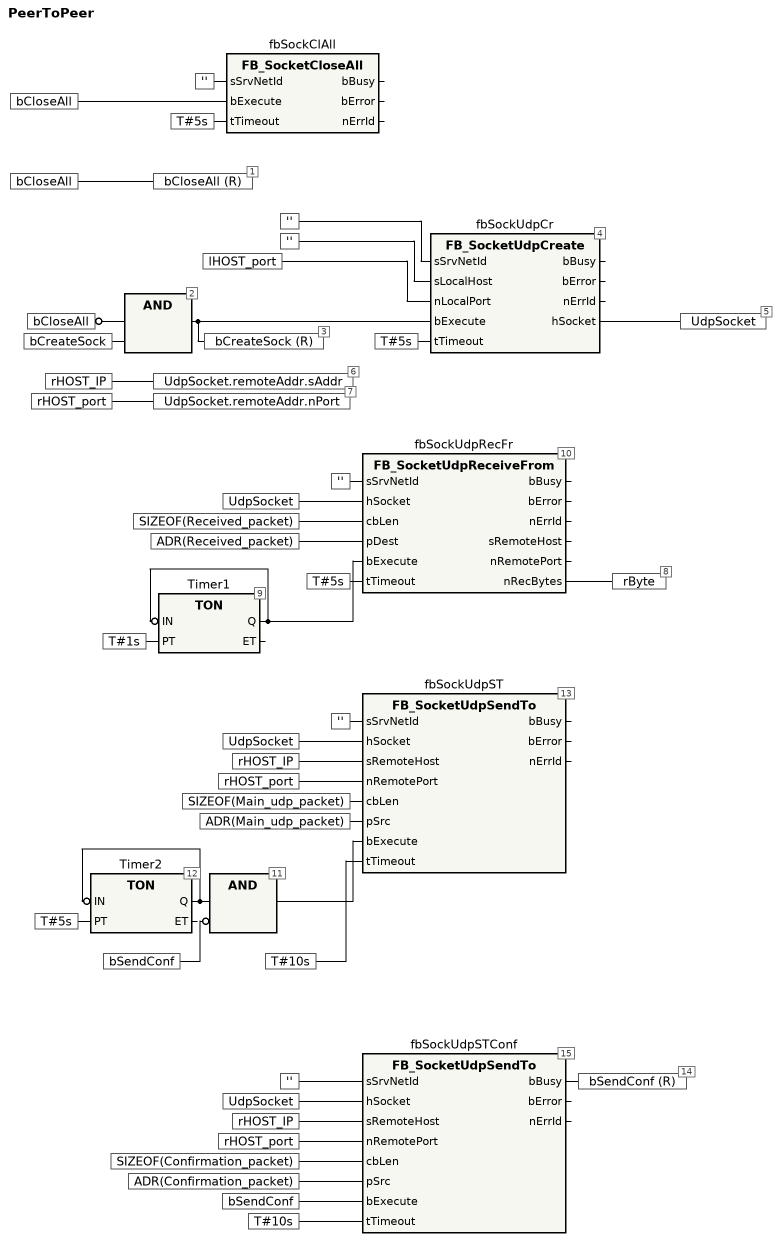
_CFC_ (* Continuous Function Chart, elements in execution order *)
#0 fbSockClAll:FB_SocketCloseAll(sSrvNetId: '', bExecute: bCloseAll, tTimeout: T#5s)
#1 R bCloseAll <= bCloseAll
#2 AND(NOT bCloseAll, bCreateSock)
#3 R bCreateSock <= #2
#4 fbSockUdpCr:FB_SocketUdpCreate(sSrvNetId: '', sLocalHost: '', nLocalPort: lHOST_port, bExecute: #2, tTimeout: T#5s)
#5 UdpSocket <= #4.hSocket
#6 UdpSocket.remoteAddr.sAddr <= rHOST_IP
#7 UdpSocket.remoteAddr.nPort <= rHOST_port
#8 rByte <= #10.nRecBytes
#9 Timer1:TON(IN: NOT #9.Q, PT: T#1s)
#10 fbSockUdpRecFr:FB_SocketUdpReceiveFrom(sSrvNetId: '', hSocket: UdpSocket, cbLen: SIZEOF(Received_packet), pDest: ADR(Received_packet), bExecute: #9.Q, tTimeout: T#5s)
#11 AND(#12.Q, NOT bSendConf)
#12 Timer2:TON(IN: NOT #12.Q, PT: T#5s)
#13 fbSockUdpST:FB_SocketUdpSendTo(sSrvNetId: '', hSocket: UdpSocket, sRemoteHost: rHOST_IP, nRemotePort: rHOST_port, cbLen: SIZEOF(Main_udp_packet), pSrc: ADR(Main_udp_packet), bExecute: #11, tTimeout: T#10s)
#14 R bSendConf <= #15.bBusy
#15 fbSockUdpSTConf:FB_SocketUdpSendTo(sSrvNetId: '', hSocket: UdpSocket, sRemoteHost: rHOST_IP, nRemotePort: rHOST_port, cbLen: SIZEOF(Confirmation_packet), pSrc: ADR(Confirmation_packet), bExecute: bSendConf, tTimeout: T#10s)
_END_CFC_
(* the same logic as Structured Text *)
fbSockClAll(sSrvNetId := '', bExecute := bCloseAll, tTimeout := T#5s);
IF bCloseAll THEN bCloseAll := FALSE; END_IF;
_t29 := NOT bCloseAll AND bCreateSock;
IF _t29 THEN bCreateSock := FALSE; END_IF;
fbSockUdpCr(sSrvNetId := '', sLocalHost := '', nLocalPort := lHOST_port, bExecute := _t29, tTimeout := T#5s);
UdpSocket := fbSockUdpCr.hSocket;
UdpSocket.remoteAddr.sAddr := rHOST_IP;
UdpSocket.remoteAddr.nPort := rHOST_port;
rByte := fbSockUdpRecFr.nRecBytes;
Timer1(IN := NOT Timer1.Q, PT := T#1s);
fbSockUdpRecFr(sSrvNetId := '', hSocket := UdpSocket, cbLen := SIZEOF(Received_packet), pDest := ADR(Received_packet), bExecute := Timer1.Q, tTimeout := T#5s);
_t76 := Timer2.Q AND NOT bSendConf;
Timer2(IN := NOT Timer2.Q, PT := T#5s);
fbSockUdpST(sSrvNetId := '', hSocket := UdpSocket, sRemoteHost := rHOST_IP, nRemotePort := rHOST_port, cbLen := SIZEOF(Main_udp_packet), pSrc := ADR(Main_udp_packet), bExecute := _t76, tTimeout := T#10s);
IF fbSockUdpSTConf.bBusy THEN bSendConf := FALSE; END_IF;
fbSockUdpSTConf(sSrvNetId := '', hSocket := UdpSocket, sRemoteHost := rHOST_IP, nRemotePort := rHOST_port, cbLen := SIZEOF(Confirmation_packet), pSrc := ADR(Confirmation_packet), bExecute := bSendConf, tTimeout := T#10s);
END_PROGRAM

(* POU Udp_receive_packet_init, ST *)
PROGRAM Udp_receive_packet_init
VAR
	Checksum_rec : WORD;
	k: INT;
	l: INT;
	i: INT;
	h: INT;
	g: INT;
	J: INT;
END_VAR
PacketSize := SIZEOF(Received_packet) - SIZEOF(Received_packet.title_packet_num) - SIZEOF(Received_packet.title_packet_code) - SIZEOF(Received_packet.title_packet_crc);
Fletcher_checksum;
Checksum_incom;
Checksum_rec := INT_TO_WORD(Received_packet.title_packet_crc);

IF (rByte> 0) THEN
IF(Checksum_rec > Checksum_incom OR Checksum_rec < Checksum_incom OR Received_packet.data_pointer > 428 OR Received_packet.data_pointer < 6) THEN
Confirmation_packet.title_packet_code := 3;
Confirmation_packet.title_packet_num := Received_packet.title_packet_num;
Confirmation_packet.title_packet_crc := Received_packet.title_packet_crc;
Confirmation_packet.data_pointer := Received_packet.data_pointer;
Confirmation_packet.data_new_value := Received_packet.data_new_value;
ELSE
Confirmation_packet.title_packet_code := 2;
Confirmation_packet.title_packet_num := Received_packet.title_packet_num;
Confirmation_packet.title_packet_crc := Received_packet.title_packet_crc;
Confirmation_packet.data_pointer := Received_packet.data_pointer;
Confirmation_packet.data_new_value := Received_packet.data_new_value;

Force_udp_packet := Main_udp_packet;
Temp_of_int[Confirmation_packet.data_pointer/2 - 2] := Confirmation_packet.data_new_value;

garage_OG_1 := INT_TO_BOOL(Force_udp_packet.grsch_garage_og[1]);
garage_OG_2 := INT_TO_BOOL(Force_udp_packet.grsch_garage_og[2]);
garage_OG_3 := INT_TO_BOOL(Force_udp_packet.grsch_garage_og[3]);
garage_OG_4 := INT_TO_BOOL(Force_udp_packet.grsch_garage_og[4]);
garage_OG_5 := INT_TO_BOOL(Force_udp_packet.grsch_garage_og[5]);
garage_OG_6 := INT_TO_BOOL(Force_udp_packet.grsch_garage_og[6]);
garage_OG_7 := INT_TO_BOOL(Force_udp_packet.grsch_garage_og[7]);
garage_OG_8 := INT_TO_BOOL(Force_udp_packet.grsch_garage_og[8]);
garage_OG_9 := INT_TO_BOOL(Force_udp_packet.grsch_garage_og[9]);
garage_OG_10 := INT_TO_BOOL(Force_udp_packet.grsch_garage_og[10]);
garage_OG_11 := INT_TO_BOOL(Force_udp_packet.grsch_garage_og[11]);
garage_OG_12 := INT_TO_BOOL(Force_udp_packet.grsch_garage_og[12]);
garage_OG_13 := INT_TO_BOOL(Force_udp_packet.grsch_garage_og[13]);
garage_OG_14 := INT_TO_BOOL(Force_udp_packet.grsch_garage_og[14]);
garage_OG_15 := INT_TO_BOOL(Force_udp_packet.grsch_garage_og[15]);
garage_OG_16 := INT_TO_BOOL(Force_udp_packet.grsch_garage_og[16]);
garage_OG_17 := INT_TO_BOOL(Force_udp_packet.grsch_garage_og[17]);
garage_OG_18 := INT_TO_BOOL(Force_udp_packet.grsch_garage_og[18]);
garage_OG_19 := INT_TO_BOOL(Force_udp_packet.grsch_garage_og[19]);
garage_OG_20 := INT_TO_BOOL(Force_udp_packet.grsch_garage_og[20]);
garage_OG_21 := INT_TO_BOOL(Force_udp_packet.grsch_garage_og[21]);
garage_OG_22 := INT_TO_BOOL(Force_udp_packet.grsch_garage_og[22]);
garage_OG_23 := INT_TO_BOOL(Force_udp_packet.grsch_garage_og[23]);
garage_OG_24 := INT_TO_BOOL(Force_udp_packet.grsch_garage_og[24]);
garage_OG_25 := INT_TO_BOOL(Force_udp_packet.grsch_garage_og[25]);
garage_OG_26 := INT_TO_BOOL(Force_udp_packet.grsch_garage_og[26]);
garage_OG_27 := INT_TO_BOOL(Force_udp_packet.grsch_garage_og[27]);
garage_OG_28 := INT_TO_BOOL(Force_udp_packet.grsch_garage_og[28]);
garage_OG_29 := INT_TO_BOOL(Force_udp_packet.grsch_garage_og[29]);
SHUF_PRESSED := INT_TO_BOOL(Force_udp_packet.grsch_SHUF_PRESSED);
PowerSystemSwitcher := INT_TO_BOOL(Force_udp_packet.grsch_power_system_switcher);
schav_force_stack  := Force_udp_packet.schav_stack;
FOR k := 1 TO 19 DO
schnog_force_stack[k] := INT_TO_BOOL(Force_udp_packet.schnog_stack[k]);
END_FOR;
FOR l := 1 TO 116 DO
schszp_force_stack[l] := INT_TO_BOOL(Force_udp_packet.schszp_stack[l]);
END_FOR;

IF (Confirmation_packet.data_pointer =  306 AND Confirmation_packet.data_new_value = 1) THEN schszp_force_stack[60] := 0; END_IF;
IF (Confirmation_packet.data_pointer =  308 AND Confirmation_packet.data_new_value = 1) THEN schszp_force_stack[61] := 0; END_IF;
IF (Confirmation_packet.data_pointer =  310 AND Confirmation_packet.data_new_value = 1) THEN schszp_force_stack[62] := 0; END_IF;
IF (Confirmation_packet.data_pointer =  312 AND Confirmation_packet.data_new_value = 1) THEN schszp_force_stack[63] := 0; END_IF;
IF (Confirmation_packet.data_pointer =  314 AND Confirmation_packet.data_new_value = 1) THEN schszp_force_stack[64] := 0; END_IF;
IF (Confirmation_packet.data_pointer =  316 AND Confirmation_packet.data_new_value = 1) THEN schszp_force_stack[55] := 0; END_IF;
IF (Confirmation_packet.data_pointer =  318 AND Confirmation_packet.data_new_value = 1) THEN schszp_force_stack[56] := 0; END_IF;
IF (Confirmation_packet.data_pointer =  320 AND Confirmation_packet.data_new_value = 1) THEN schszp_force_stack[57] := 0; END_IF;
IF (Confirmation_packet.data_pointer =  322 AND Confirmation_packet.data_new_value = 1) THEN schszp_force_stack[58] := 0; END_IF;
IF (Confirmation_packet.data_pointer =  324 AND Confirmation_packet.data_new_value = 1) THEN schszp_force_stack[59] := 0; END_IF;

END_IF;
IF(J = 0) THEN
bSendConf := TRUE;
END_IF;
J := J + 1;
END_IF;

IF(rByte = 0) THEN
J := 0;
END_IF;
END_PROGRAM

(* POU AutoReset, CFC *)
PROGRAM AutoReset
VAR
	AutoResetCX: PLC_Reset;
	AutoStartCX: PLC_Start;
END_VAR
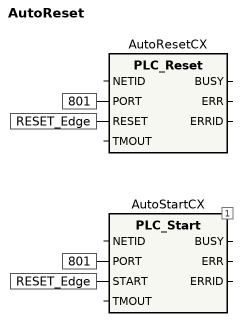
_CFC_ (* Continuous Function Chart, elements in execution order *)
#0 AutoResetCX:PLC_Reset(NETID: -, PORT: 801, RESET: RESET_Edge, TMOUT: -)
#1 AutoStartCX:PLC_Start(NETID: -, PORT: 801, START: RESET_Edge, TMOUT: -)
_END_CFC_
(* the same logic as Structured Text *)
AutoResetCX(PORT := 801, RESET := RESET_Edge);
AutoStartCX(PORT := 801, START := RESET_Edge);
END_PROGRAM

(* POU CalcPower, ST *)
PROGRAM CalcPower
VAR
	koef_power: REAL := 0.5;
	koef_voltage: REAL := 0.1;
	koef_current: REAL := 0.005;
END_VAR
KL3403_1_P :=ABS(KL3403_1_P1 + KL3403_1_P2 + KL3403_1_P3)*koef_power/1000;
KL3403_2_P :=ABS (KL3403_2_P1 + KL3403_2_P2 + KL3403_2_P3)*koef_power/1000;
KL3403_3_P := ABS(KL3403_3_P1 + KL3403_3_P2 + KL3403_3_P3)*koef_power/1000;
KL3403_4_P := ABS(KL3403_4_P1 + KL3403_4_P2 + KL3403_4_P3)*koef_power/1000;
KL3403_5_P := ABS(KL3403_5_P1 + KL3403_5_P2 + KL3403_5_P3)*koef_power/1000;

KL3403_1_V :=ABS(KL3403_1_P1 + KL3403_1_P2 + KL3403_1_P3)*koef_voltage/3;
KL3403_2_V :=ABS (KL3403_2_P1 + KL3403_2_P2 + KL3403_2_P3)*koef_voltage/3;
KL3403_3_V := ABS(KL3403_3_P1 + KL3403_3_P2 + KL3403_3_P3)*koef_voltage/3;
KL3403_4_V := ABS(KL3403_4_P1 + KL3403_4_P2 + KL3403_4_P3)*koef_voltage/3;
KL3403_5_V := ABS(KL3403_5_P1 + KL3403_5_P2 + KL3403_5_P3)*koef_voltage/3;

KL3403_1_I :=ABS(KL3403_1_P1 + KL3403_1_P2 + KL3403_1_P3)*koef_current/3;
KL3403_2_I :=ABS (KL3403_2_P1 + KL3403_2_P2 + KL3403_2_P3)*koef_current/3;
KL3403_3_I := ABS(KL3403_3_P1 + KL3403_3_P2 + KL3403_3_P3)*koef_current/3;
KL3403_4_I := ABS(KL3403_4_P1 + KL3403_4_P2 + KL3403_4_P3)*koef_current/3;
KL3403_5_I := ABS(KL3403_5_P1 + KL3403_5_P2 + KL3403_5_P3)*koef_current/3;
END_PROGRAM

(* POU CheckLight, CFC *)
PROGRAM CheckLight
VAR

	ADSWRITE: FW_AdsWrite;
	timer: TON;
	ttimer1: TOF;
	timer2: TON;

	AdsWriteLandscape: FW_AdsWrite;
	timer2l: TON;
	timer22: TON;
	AdsWriteNight: FW_AdsWrite;
	timer23: TON;
	AdsWriteUOG: FW_AdsWrite;
	timer24: TON;
	ADSnew222: ADSWRITE;
END_VAR
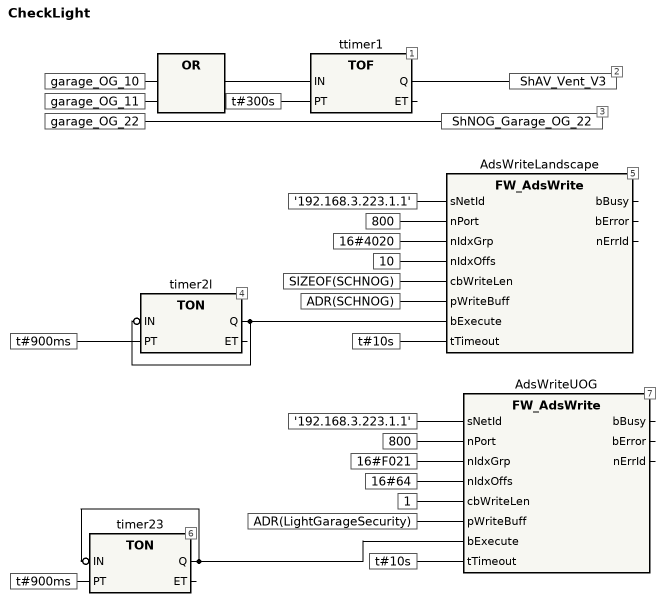
_CFC_ (* Continuous Function Chart, elements in execution order *)
#0 OR(garage_OG_10, garage_OG_11)
#1 ttimer1:TOF(IN: #0, PT: t#300s)
#2 ShAV_Vent_V3 <= #1.Q
#3 ShNOG_Garage_OG_22 <= garage_OG_22
#4 timer2l:TON(IN: NOT #4.Q, PT: t#900ms)
#5 AdsWriteLandscape:FW_AdsWrite(sNetId: '192.168.3.223.1.1', nPort: 800, nIdxGrp: 16#4020, nIdxOffs: 10, cbWriteLen: SIZEOF(SCHNOG), pWriteBuff: ADR(SCHNOG), bExecute: #4.Q, tTimeout: t#10s)
#6 timer23:TON(IN: NOT #6.Q, PT: t#900ms)
#7 AdsWriteUOG:FW_AdsWrite(sNetId: '192.168.3.223.1.1', nPort: 800, nIdxGrp: 16#F021, nIdxOffs: 16#64, cbWriteLen: 1, pWriteBuff: ADR(LightGarageSecurity), bExecute: #6.Q, tTimeout: t#10s)
_END_CFC_
(* the same logic as Structured Text *)
ttimer1(IN := garage_OG_10 OR garage_OG_11, PT := t#300s);
ShAV_Vent_V3 := ttimer1.Q;
ShNOG_Garage_OG_22 := garage_OG_22;
timer2l(IN := NOT timer2l.Q, PT := t#900ms);
AdsWriteLandscape(sNetId := '192.168.3.223.1.1', nPort := 800, nIdxGrp := 16#4020, nIdxOffs := 10, cbWriteLen := SIZEOF(SCHNOG), pWriteBuff := ADR(SCHNOG), bExecute := timer2l.Q, tTimeout := t#10s);
timer23(IN := NOT timer23.Q, PT := t#900ms);
AdsWriteUOG(sNetId := '192.168.3.223.1.1', nPort := 800, nIdxGrp := 16#F021, nIdxOffs := 16#64, cbWriteLen := 1, pWriteBuff := ADR(LightGarageSecurity), bExecute := timer23.Q, tTimeout := t#10s);
END_PROGRAM

(* POU ReadADS, CFC *)
PROGRAM ReadADS
VAR
	ReadADS: FW_AdsRead;
	timer2: TON;

	bBusy		: BOOL;
	bError		: BOOL;
	nErrId		: UDINT;
	cbRead		: UDINT;


	bBusy2			: BOOL;
	bError2			: BOOL;
	nErrId2			: UDINT;
	cbRead2		: UDINT;

	ReadLights: FW_AdsRead;
	timer3: TON;
	timer32: TON;
	bBusy3: BOOL;
	bError3: BOOL;
	ReadSCHAV: FW_AdsRead;
	SchAV_Muhamed: FW_AdsWrite;
END_VAR
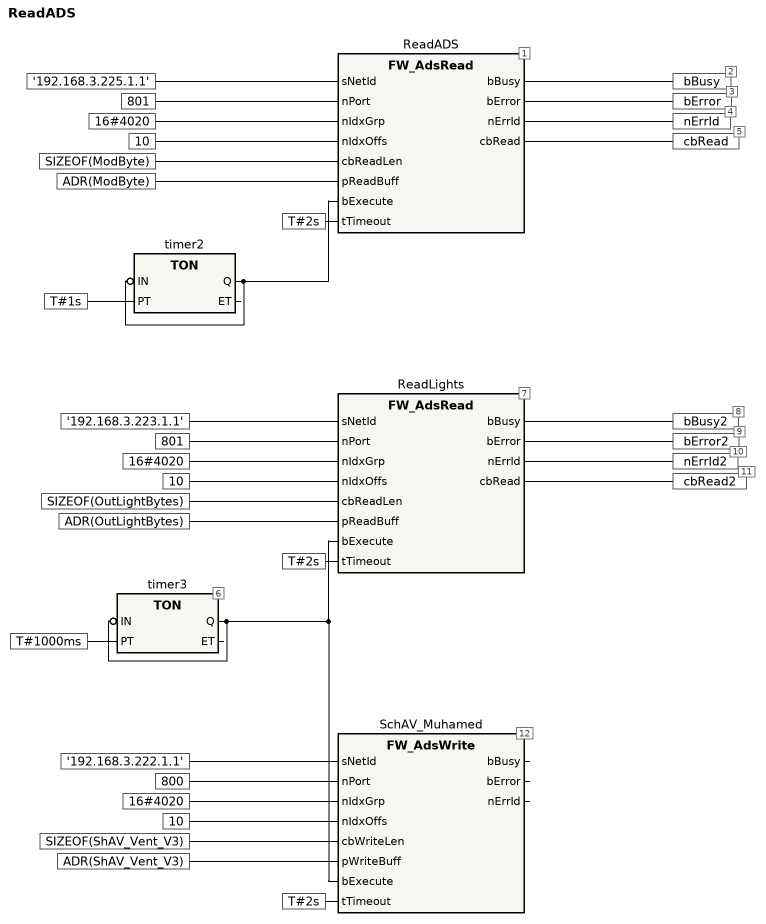
_CFC_ (* Continuous Function Chart, elements in execution order *)
#0 timer2:TON(IN: NOT #0.Q, PT: T#1s)
#1 ReadADS:FW_AdsRead(sNetId: '192.168.3.225.1.1', nPort: 801, nIdxGrp: 16#4020, nIdxOffs: 10, cbReadLen: SIZEOF(ModByte), pReadBuff: ADR(ModByte), bExecute: #0.Q, tTimeout: T#2s)
#2 bBusy <= #1.bBusy
#3 bError <= #1.bError
#4 nErrId <= #1.nErrId
#5 cbRead <= #1.cbRead
#6 timer3:TON(IN: NOT #6.Q, PT: T#1000ms)
#7 ReadLights:FW_AdsRead(sNetId: '192.168.3.223.1.1', nPort: 801, nIdxGrp: 16#4020, nIdxOffs: 10, cbReadLen: SIZEOF(OutLightBytes), pReadBuff: ADR(OutLightBytes), bExecute: #6.Q, tTimeout: T#2s)
#8 bBusy2 <= #7.bBusy
#9 bError2 <= #7.bError
#10 nErrId2 <= #7.nErrId
#11 cbRead2 <= #7.cbRead
#12 SchAV_Muhamed:FW_AdsWrite(sNetId: '192.168.3.222.1.1', nPort: 800, nIdxGrp: 16#4020, nIdxOffs: 10, cbWriteLen: SIZEOF(ShAV_Vent_V3), pWriteBuff: ADR(ShAV_Vent_V3), bExecute: #6.Q, tTimeout: T#2s)
_END_CFC_
(* the same logic as Structured Text *)
timer2(IN := NOT timer2.Q, PT := T#1s);
ReadADS(sNetId := '192.168.3.225.1.1', nPort := 801, nIdxGrp := 16#4020, nIdxOffs := 10, cbReadLen := SIZEOF(ModByte), pReadBuff := ADR(ModByte), bExecute := timer2.Q, tTimeout := T#2s);
bBusy := ReadADS.bBusy;
bError := ReadADS.bError;
nErrId := ReadADS.nErrId;
cbRead := ReadADS.cbRead;
timer3(IN := NOT timer3.Q, PT := T#1000ms);
ReadLights(sNetId := '192.168.3.223.1.1', nPort := 801, nIdxGrp := 16#4020, nIdxOffs := 10, cbReadLen := SIZEOF(OutLightBytes), pReadBuff := ADR(OutLightBytes), bExecute := timer3.Q, tTimeout := T#2s);
bBusy2 := ReadLights.bBusy;
bError2 := ReadLights.bError;
nErrId2 := ReadLights.nErrId;
cbRead2 := ReadLights.cbRead;
SchAV_Muhamed(sNetId := '192.168.3.222.1.1', nPort := 800, nIdxGrp := 16#4020, nIdxOffs := 10, cbWriteLen := SIZEOF(ShAV_Vent_V3), pWriteBuff := ADR(ShAV_Vent_V3), bExecute := timer3.Q, tTimeout := T#2s);
END_PROGRAM

(* Visualisation CURRENTPAGE
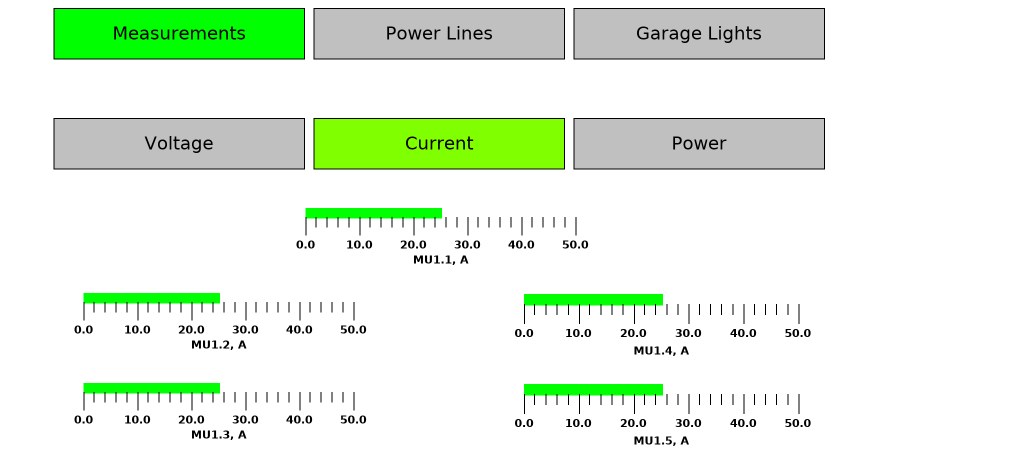
rounded rectangle at (10,130)-(261,181): text "Voltage"; taps KoefV; opens VoltagePage
rounded rectangle at (270,130)-(521,181): text "Current"
rounded rectangle at (530,130)-(781,181): text "Power"; taps KoefP; opens PowerPage
group at (460,290)-(771,381)
  rectangle at (0,0)-(1,1): text "{ExtendedElement},Visu\ElementDLL.ete,1,@Bargraph,311,91,0,0,0,KL3403_4_I,MU1.4, A,%.1f,2,10,0,50,0,0,0,0,0,0,0,-13,16,700,Arial,0,255,0,255,0,0,0,0,0,0,0,"
  rectangle at (20,15)-(156,25): alarm colour if (KL3403_4_I) < 0; right ((KL3403_4_I * 1.0) - 25)  * 5.4
  rectangle at (8,44)-(32,84): text "0.0"
  rectangle at (57,44)-(90,84): text "10.0"
  rectangle at (111,44)-(144,84): text "20.0"
  rectangle at (165,44)-(198,84): text "30.0"
  rectangle at (219,44)-(252,84): text "40.0"
  rectangle at (273,44)-(306,84): text "50.0"
  rectangle at (100,59)-(210,75): text "MU1.4, A"
group at (460,380)-(771,471)
  rectangle at (0,0)-(1,1): text "{ExtendedElement},Visu\ElementDLL.ete,1,@Bargraph,311,91,0,0,0,KL3403_5_I,MU1.5, A,%.1f,2,10,0,50,0,0,0,0,0,0,0,-13,16,700,Arial,0,255,0,255,0,0,0,0,0,0,0,"
  rectangle at (20,15)-(156,25): alarm colour if (KL3403_5_I) < 0; right ((KL3403_5_I * 1.0) - 25)  * 5.4
  rectangle at (8,44)-(32,84): text "0.0"
  rectangle at (57,44)-(90,84): text "10.0"
  rectangle at (111,44)-(144,84): text "20.0"
  rectangle at (165,44)-(198,84): text "30.0"
  rectangle at (219,44)-(252,84): text "40.0"
  rectangle at (273,44)-(306,84): text "50.0"
  rectangle at (100,59)-(210,75): text "MU1.5, A"
rounded rectangle at (10,20)-(261,71): text "Measurements"
rounded rectangle at (270,20)-(521,71): text "Power Lines"; opens MainPage
rounded rectangle at (530,20)-(781,71): text "Garage Lights"; opens GarageLight
group at (28,305)-(326,374)
  rectangle at (12,0)-(148,10): alarm colour if (KL3403_1_I) < 0; right ((KL3403_1_I * 1.0) - 25)  * 5.4
  rectangle at (0,29)-(24,69): text "0.0"
  rectangle at (49,29)-(82,69): text "10.0"
  rectangle at (103,29)-(136,69): text "20.0"
  rectangle at (157,29)-(190,69): text "30.0"
  rectangle at (211,29)-(244,69): text "40.0"
  rectangle at (265,29)-(298,69): text "50.0"
  rectangle at (92,44)-(202,60): text "MU1.2, A"
group at (28,395)-(326,464)
  rectangle at (12,0)-(148,10): alarm colour if (KL3403_2_I) < 0; right ((KL3403_2_I * 1.0) - 25)  * 5.4
  rectangle at (0,29)-(24,69): text "0.0"
  rectangle at (49,29)-(82,69): text "10.0"
  rectangle at (103,29)-(136,69): text "20.0"
  rectangle at (157,29)-(190,69): text "30.0"
  rectangle at (211,29)-(244,69): text "40.0"
  rectangle at (265,29)-(298,69): text "50.0"
  rectangle at (92,44)-(202,60): text "MU1.3, A"
group at (250,220)-(548,289)
  rectangle at (12,0)-(148,10): alarm colour if (KL3403_3_I) < 0; right ((KL3403_3_I * 1.0) - 25)  * 5.4
  rectangle at (0,29)-(24,69): text "0.0"
  rectangle at (49,29)-(82,69): text "10.0"
  rectangle at (103,29)-(136,69): text "20.0"
  rectangle at (157,29)-(190,69): text "30.0"
  rectangle at (211,29)-(244,69): text "40.0"
  rectangle at (265,29)-(298,69): text "50.0"
  rectangle at (92,44)-(202,60): text "MU1.1, A"
130 more shapes without text or variables
*)

(* Visualisation GARAGELIGHT
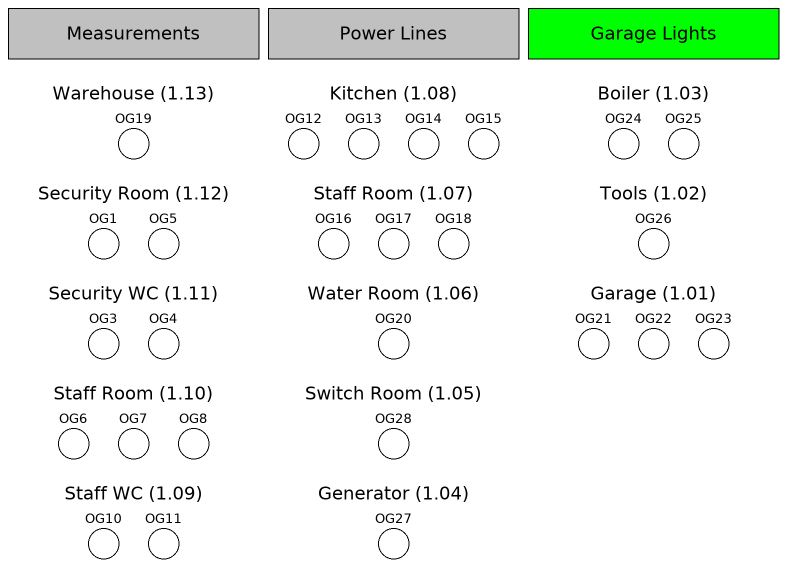
rectangle at (10,190)-(261,221): text "Security Room (1.12)"
ellipse at (90,240)-(121,271): alarm colour if garage_OG_1; toggles Garage_OG_1
ellipse at (150,240)-(181,271): alarm colour if garage_OG_5
rectangle at (80,220)-(131,241): text "OG1"
rectangle at (140,220)-(191,241): text "OG5"
ellipse at (120,140)-(151,171): alarm colour if garage_OG_19
rectangle at (110,120)-(161,141): text "OG19"
rectangle at (10,90)-(261,121): text "Warehouse (1.13)"
rectangle at (10,290)-(261,321): text "Security WC (1.11)"
ellipse at (90,340)-(121,371): alarm colour if garage_OG_3
ellipse at (150,340)-(181,371): alarm colour if garage_OG_4
rectangle at (80,320)-(131,341): text "OG3"
rectangle at (140,320)-(191,341): text "OG4"
rectangle at (10,490)-(261,521): text "Staff WC (1.09)"
ellipse at (90,540)-(121,571): alarm colour if garage_OG_10
ellipse at (150,540)-(181,571): alarm colour if garage_OG_11
rectangle at (80,520)-(131,541): text "OG10"
rectangle at (140,520)-(191,541): text "OG11"
rectangle at (10,390)-(261,421): text "Staff Room (1.10)"
ellipse at (60,440)-(91,471): alarm colour if garage_OG_6
ellipse at (120,440)-(151,471): alarm colour if garage_OG_7
rectangle at (50,420)-(101,441): text "OG6"
rectangle at (110,420)-(161,441): text "OG7"
ellipse at (180,440)-(211,471): alarm colour if garage_OG_8
rectangle at (170,420)-(221,441): text "OG8"
rectangle at (270,90)-(521,121): text "Kitchen (1.08)"
ellipse at (290,140)-(321,171): alarm colour if garage_OG_12
ellipse at (350,140)-(381,171): alarm colour if garage_OG_13
rectangle at (280,120)-(331,141): text "OG12"
rectangle at (340,120)-(391,141): text "OG13"
rectangle at (270,190)-(521,221): text "Staff Room (1.07)"
rectangle at (270,290)-(521,321): text "Water Room (1.06)"
ellipse at (380,340)-(411,371): alarm colour if garage_OG_20
rectangle at (370,320)-(421,341): text "OG20"
rectangle at (270,490)-(521,521): text "Generator (1.04)"
ellipse at (380,540)-(411,571): alarm colour if garage_OG_27
rectangle at (370,520)-(421,541): text "OG27"
rectangle at (270,390)-(521,421): text "Switch Room (1.05)"
ellipse at (380,440)-(411,471): alarm colour if garage_OG_28; toggles Garage_OG_28
rectangle at (370,420)-(421,441): text "OG28"
ellipse at (410,140)-(441,171): alarm colour if garage_OG_14
ellipse at (470,140)-(501,171): alarm colour if garage_OG_15
rectangle at (400,120)-(451,141): text "OG14"
rectangle at (460,120)-(511,141): text "OG15"
ellipse at (320,240)-(351,271): alarm colour if garage_OG_16
ellipse at (380,240)-(411,271): alarm colour if garage_OG_17
rectangle at (310,220)-(361,241): text "OG16"
rectangle at (370,220)-(421,241): text "OG17"
ellipse at (440,240)-(471,271): alarm colour if garage_OG_18
rectangle at (430,220)-(481,241): text "OG18"
rectangle at (530,90)-(781,121): text "Boiler (1.03)"
rectangle at (530,190)-(781,221): text "Tools (1.02)"
rectangle at (530,290)-(781,321): text "Garage (1.01)"
ellipse at (610,140)-(641,171): alarm colour if garage_OG_24
ellipse at (670,140)-(701,171): alarm colour if garage_OG_25
rectangle at (600,120)-(651,141): text "OG24"
rectangle at (660,120)-(711,141): text "OG25"
ellipse at (640,240)-(671,271): alarm colour if garage_OG_26
rectangle at (630,220)-(681,241): text "OG26"
ellipse at (580,340)-(611,371): alarm colour if garage_OG_21
ellipse at (640,340)-(671,371): alarm colour if garage_OG_22
rectangle at (570,320)-(621,341): text "OG21"
rectangle at (630,320)-(681,341): text "OG22"
ellipse at (700,340)-(731,371): alarm colour if garage_OG_23
rectangle at (690,320)-(741,341): text "OG23"
rounded rectangle at (10,20)-(261,71): text "Measurements"; opens PowerPage
rounded rectangle at (270,20)-(521,71): text "Power Lines"; opens MainPage
rounded rectangle at (530,20)-(781,71): text "Garage Lights"
*)

(* Visualisation MAINPAGE
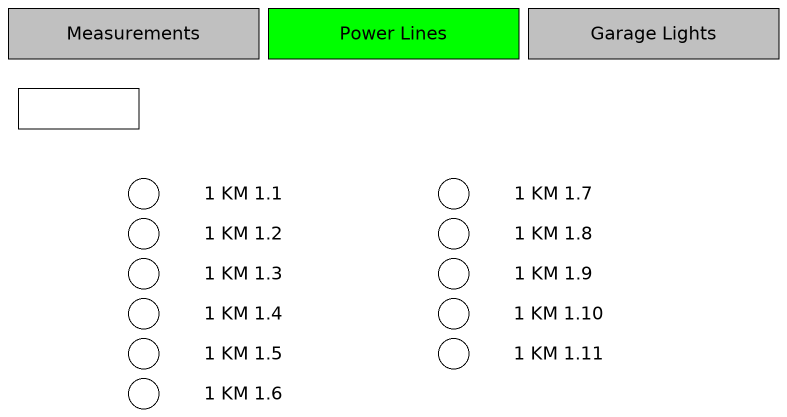
ellipse at (130,190)-(161,221): alarm colour if power_VRU_switch[1]; runs INTERN ASSIGN SHUF_PRESSED:=(TRUE)
ellipse at (130,270)-(161,301): alarm colour if power_VRU_switch[3]; runs INTERN ASSIGN SHUF_PRESSED:=(TRUE)
ellipse at (130,310)-(161,341): alarm colour if power_VRU_switch[4]; runs INTERN ASSIGN SHUF_PRESSED:=(TRUE)
ellipse at (130,350)-(161,381): alarm colour if power_VRU_switch[5]; runs INTERN ASSIGN SHUF_PRESSED:=(TRUE)
ellipse at (130,390)-(161,421): alarm colour if power_VRU_switch[6]; runs INTERN ASSIGN SHUF_PRESSED:=(TRUE)
ellipse at (440,230)-(471,261): alarm colour if power_VRU_switch[8]; runs INTERN ASSIGN SHUF_PRESSED:=(TRUE)
ellipse at (440,190)-(471,221): alarm colour if power_VRU_switch[7]; runs INTERN ASSIGN SHUF_PRESSED:=(TRUE)
ellipse at (440,270)-(471,301): alarm colour if power_VRU_switch[9]; runs INTERN ASSIGN SHUF_PRESSED:=(TRUE)
ellipse at (440,310)-(471,341): alarm colour if power_VRU_switch[10]; runs INTERN ASSIGN SHUF_PRESSED:=(TRUE)
ellipse at (130,230)-(161,261): alarm colour if power_VRU_switch[2]; runs INTERN ASSIGN SHUF_PRESSED:=(TRUE)
rectangle at (170,230)-(321,261): text "1 KM 1.2"
rectangle at (180,190)-(311,221): text "1 KM 1.1"
rectangle at (170,350)-(321,381): text "1 KM 1.5"
rectangle at (170,390)-(321,421): text "1 KM 1.6"
rectangle at (480,190)-(631,221): text "1 KM 1.7"
rectangle at (170,270)-(321,301): text "1 KM 1.3"
rectangle at (170,310)-(321,341): text "1 KM 1.4"
rectangle at (480,230)-(631,261): text "1 KM 1.8"
rectangle at (480,270)-(631,301): text "1 KM 1.9"
rectangle at (490,350)-(631,381): text "1 KM 1.11"
rounded rectangle at (10,20)-(261,71): text "Measurements"; opens PowerPage
rounded rectangle at (270,20)-(521,71): text "Power Lines"
rounded rectangle at (530,20)-(781,71): text "Garage Lights"; opens GarageLight
ellipse at (440,350)-(471,381): alarm colour if power_VRU_switch[11]; runs INTERN ASSIGN SHUF_PRESSED:=(TRUE)
rectangle at (490,310)-(631,341): text "1 KM 1.10"
rectangle at (20,100)-(141,141): alarm colour if PowerSystemSwitcher; toggles PowerSystemSwitcher
*)

(* Visualisation POWERPAGE
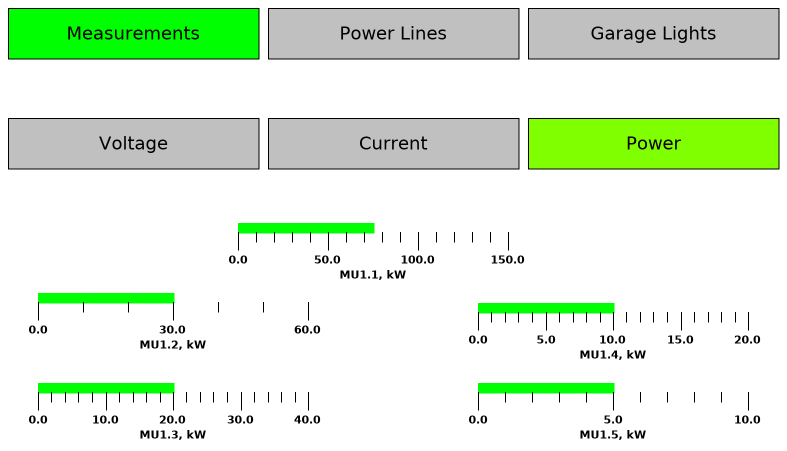
rounded rectangle at (10,130)-(261,181): text "Voltage"; taps KoefV; opens VoltagePage
rounded rectangle at (270,130)-(521,181): text "Current"; taps KoefI; opens CurrentPage
rounded rectangle at (530,130)-(781,181): text "Power"
rounded rectangle at (10,20)-(261,71): text "Measurements"
rounded rectangle at (270,20)-(521,71): text "Power Lines"; opens MainPage
rounded rectangle at (530,20)-(781,71): text "Garage Lights"; opens GarageLight
group at (228,235)-(531,304)
  rectangle at (12,0)-(148,10): alarm colour if (KL3403_3_P) < 0; right ((KL3403_3_P * 1.0) - 75)  * 1.8
  rectangle at (0,29)-(24,69): text "0.0"
  rectangle at (85,29)-(118,69): text "50.0"
  rectangle at (170,29)-(213,69): text "100.0"
  rectangle at (260,29)-(303,69): text "150.0"
  rectangle at (81,44)-(213,60): text "MU1.1, kW"
group at (28,305)-(326,374)
  rectangle at (12,0)-(148,10): alarm colour if (KL3403_1_P) < 0; right ((KL3403_1_P * 1.0) - 30)  * 4.5
  rectangle at (0,29)-(24,69): text "0.0"
  rectangle at (130,29)-(163,69): text "30.0"
  rectangle at (265,29)-(298,69): text "60.0"
  rectangle at (81,44)-(213,60): text "MU1.2, kW"
group at (28,395)-(326,464)
  rectangle at (12,0)-(148,10): alarm colour if (KL3403_2_P) < 0; right ((KL3403_2_P * 1.0) - 20)  * 6.75
  rectangle at (0,29)-(24,69): text "0.0"
  rectangle at (63,29)-(96,69): text "10.0"
  rectangle at (130,29)-(163,69): text "20.0"
  rectangle at (198,29)-(231,69): text "30.0"
  rectangle at (265,29)-(298,69): text "40.0"
  rectangle at (81,44)-(213,60): text "MU1.3, kW"
group at (468,315)-(766,384)
  rectangle at (12,0)-(148,10): alarm colour if (KL3403_4_P) < 0; right ((KL3403_4_P * 1.0) - 10)  * 13.5
  rectangle at (0,29)-(24,69): text "0.0"
  rectangle at (68,29)-(92,69): text "5.0"
  rectangle at (130,29)-(163,69): text "10.0"
  rectangle at (198,29)-(231,69): text "15.0"
  rectangle at (265,29)-(298,69): text "20.0"
  rectangle at (81,44)-(213,60): text "MU1.4, kW"
group at (468,395)-(766,464)
  rectangle at (12,0)-(148,10): alarm colour if (KL3403_5_P) < 0; right ((KL3403_5_P * 1.0) - 5)  * 27
  rectangle at (0,29)-(24,69): text "0.0"
  rectangle at (135,29)-(159,69): text "5.0"
  rectangle at (265,29)-(298,69): text "10.0"
  rectangle at (81,44)-(213,60): text "MU1.5, kW"
76 more shapes without text or variables
*)

(* Visualisation VOLTAGEPAGE
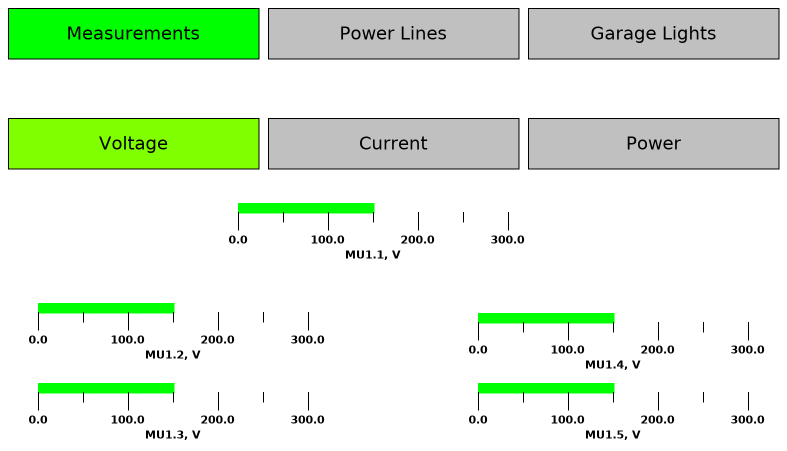
rounded rectangle at (10,130)-(261,181): text "Voltage"
rounded rectangle at (270,130)-(521,181): text "Current"; taps KoefI; opens CurrentPage
rounded rectangle at (530,130)-(781,181): text "Power"; taps KoefP; opens PowerPage
rounded rectangle at (10,20)-(261,71): text "Measurements"
rounded rectangle at (270,20)-(521,71): text "Power Lines"; opens MainPage
rounded rectangle at (530,20)-(781,71): text "Garage Lights"; opens GarageLight
group at (228,215)-(531,284)
  rectangle at (12,0)-(148,10): alarm colour if (KL3403_3_V) < 0; right ((KL3403_3_V * 1.0) - 150)  * 0.9
  rectangle at (0,29)-(24,69): text "0.0"
  rectangle at (80,29)-(123,69): text "100.0"
  rectangle at (170,29)-(213,69): text "200.0"
  rectangle at (260,29)-(303,69): text "300.0"
  rectangle at (92,44)-(202,60): text "MU1.1, V"
group at (28,315)-(331,384)
  rectangle at (12,0)-(148,10): alarm colour if (KL3403_1_V) < 0; right ((KL3403_1_V * 1.0) - 150)  * 0.9
  rectangle at (0,29)-(24,69): text "0.0"
  rectangle at (80,29)-(123,69): text "100.0"
  rectangle at (170,29)-(213,69): text "200.0"
  rectangle at (260,29)-(303,69): text "300.0"
  rectangle at (92,44)-(202,60): text "MU1.2, V"
group at (28,395)-(331,464)
  rectangle at (12,0)-(148,10): alarm colour if (KL3403_1_V) < 0; right ((KL3403_2_V * 1.0) - 150)  * 0.9
  rectangle at (0,29)-(24,69): text "0.0"
  rectangle at (80,29)-(123,69): text "100.0"
  rectangle at (170,29)-(213,69): text "200.0"
  rectangle at (260,29)-(303,69): text "300.0"
  rectangle at (92,44)-(202,60): text "MU1.3, V"
group at (468,325)-(771,394)
  rectangle at (12,0)-(148,10): alarm colour if (KL3403_4_V) < 0; right ((KL3403_4_V * 1.0) - 150)  * 0.9
  rectangle at (0,29)-(24,69): text "0.0"
  rectangle at (80,29)-(123,69): text "100.0"
  rectangle at (170,29)-(213,69): text "200.0"
  rectangle at (260,29)-(303,69): text "300.0"
  rectangle at (92,44)-(202,60): text "MU1.4, V"
group at (468,395)-(771,464)
  rectangle at (12,0)-(148,10): alarm colour if (KL3403_5_V) < 0; right ((KL3403_5_V * 1.0) - 150)  * 0.9
  rectangle at (0,29)-(24,69): text "0.0"
  rectangle at (80,29)-(123,69): text "100.0"
  rectangle at (170,29)-(213,69): text "200.0"
  rectangle at (260,29)-(303,69): text "300.0"
  rectangle at (92,44)-(202,60): text "MU1.5, V"
35 more shapes without text or variables
*)
